// TIA Portal V20 export
DATA_BLOCK "ControlNodes"   // DB83
{ DB_Accessible_From_OPC_UA := 'FALSE' }
AUTHOR : ERsystem_FA2_DH. Kim
// stored: DBAccessibleFromOPCUA false, DBAccessibleFromWebserver false, MemoryReserve 100, Namespace Unit1.Em6
   VAR
      em { ExternalWritable := 'False'} : "LAF_typeEmControlNode";
      cm : Struct
         Interlock : Struct
            finalRollerFrontAxisX : "LER_typeAxisInterlock";
            finalRollerRearAxisX : "LER_typeAxisInterlock";
            mendrelAnodeFrontAxisY : "LER_typeAxisInterlock";
            mendrelAnodeFrontAxisZ : "LER_typeAxisInterlock";
            mendrelAnodeRearAxisY : "LER_typeAxisInterlock";
            mendrelAnodeRearAxisZ : "LER_typeAxisInterlock";
            mendrelCathodeFrontAxisY : "LER_typeAxisInterlock";
            mendrelCathodeFrontAxisZ : "LER_typeAxisInterlock";
            mendrelCathodeRearAxisY : "LER_typeAxisInterlock";
            mendrelCathodeRearAxisZ : "LER_typeAxisInterlock";
            stackTableAxisZ : "LER_typeAxisInterlock";
            stackTableOutFrontAxisZ : "LER_typeAxisInterlock";
            stackTableOutRearAxisZ : "LER_typeAxisInterlock";
            mendrelAnodeFrontClamp : "LER_typeTwoWayActInterlock";
            mendrelAnodeRearClamp : "LER_typeTwoWayActInterlock";
            mendrelCathodeFrontClamp : "LER_typeTwoWayActInterlock";
            mendrelCathodeRearClamp : "LER_typeTwoWayActInterlock";
            stackTableVaccum : "LER_typeTwoWayActInterlock";
            StackTableGapPadUpDown : "LER_typeTwoWayActInterlock";
         END_STRUCT;
         Command : Struct
            finalRollerFrontAxisX { S7_SetPoint := 'True'} : "LER_typeAxisCommand";
            finalRollerRearAxisX { S7_SetPoint := 'True'} : "LER_typeAxisCommand";
            mendrelAnodeFrontAxisY { S7_SetPoint := 'True'} : "LER_typeAxisCommand";
            mendrelAnodeFrontAxisZ { S7_SetPoint := 'True'} : "LER_typeAxisCommand";
            mendrelAnodeRearAxisY { S7_SetPoint := 'True'} : "LER_typeAxisCommand";
            mendrelAnodeRearAxisZ { S7_SetPoint := 'True'} : "LER_typeAxisCommand";
            mendrelCathodeFrontAxisY { S7_SetPoint := 'True'} : "LER_typeAxisCommand";
            mendrelCathodeFrontAxisZ { S7_SetPoint := 'True'} : "LER_typeAxisCommand";
            mendrelCathodeRearAxisY { S7_SetPoint := 'True'} : "LER_typeAxisCommand";
            mendrelCathodeRearAxisZ { S7_SetPoint := 'True'} : "LER_typeAxisCommand";
            stackTableAxisZ { S7_SetPoint := 'True'} : "LER_typeAxisCommand";
            stackTableOutFrontAxisZ { S7_SetPoint := 'True'} : "LER_typeAxisCommand";
            stackTableOutRearAxisZ { S7_SetPoint := 'True'} : "LER_typeAxisCommand";
         END_STRUCT;
         softCam { S7_SetPoint := 'True'} : "Unit1.type_emRelations_em6_SoftCam";
         brakeTest : Struct
            mendrelAnodeFrontAxisZ : "LER_typeBrakeTestEmControlNoeds";
            mendrelAnodeRearAxisZ : "LER_typeBrakeTestEmControlNoeds";
            mendrelCathodeFrontAxisZ : "LER_typeBrakeTestEmControlNoeds";
            mendrelCathodeRearAxisZ : "LER_typeBrakeTestEmControlNoeds";
            stackTableAxisZ : "LER_typeBrakeTestEmControlNoeds";
            stackTableOutFrontAxisZ : "LER_typeBrakeTestEmControlNoeds";
            stackTableOutRearAxisZ : "LER_typeBrakeTestEmControlNoeds";
         END_STRUCT;
         gearIn : Struct
            finalRollerAxisX : "LER_typeGearInControlNodes";
            stackTableOutAxisZ : "LER_typeGearInControlNodes";
            finalRollerFrontAxisX : Struct
               Execute : Bool;
               ContinuousUpdate : Bool;
               RatioNumerator : DInt;
               RatioDenominator : DInt;
               Acceleration : LReal;
               Deceleration : LReal;
               Jerk : LReal;
               PositionControlled : Bool;
               StartSync : Bool;
               InSync : Bool;
               ContinuousUpdateActive : Bool;
               Busy : Bool;
               CommandAborted : Bool;
               Error : Bool;
               ErrorId : Word;
            END_STRUCT;
            finalRollerRearAxisX : Struct
               Execute : Bool;
               ContinuousUpdate : Bool;
               RatioNumerator : DInt;
               RatioDenominator : DInt;
               Acceleration : LReal;
               Deceleration : LReal;
               Jerk : LReal;
               PositionControlled : Bool;
               StartSync : Bool;
               InSync : Bool;
               ContinuousUpdateActive : Bool;
               Busy : Bool;
               CommandAborted : Bool;
               Error : Bool;
               ErrorId : Word;
            END_STRUCT;
            stackTableOutFrontAxisZ : Struct
               Execute : Bool;
               ContinuousUpdate : Bool;
               RatioNumerator : DInt;
               RatioDenominator : DInt;
               Acceleration : LReal;
               Deceleration : LReal;
               Jerk : LReal;
               PositionControlled : Bool;
               StartSync : Bool;
               InSync : Bool;
               ContinuousUpdateActive : Bool;
               Busy : Bool;
               CommandAborted : Bool;
               Error : Bool;
               ErrorId : Word;
            END_STRUCT;
            stackTableOutRearAxisZ : Struct
               Execute : Bool;
               ContinuousUpdate : Bool;
               RatioNumerator : DInt;
               RatioDenominator : DInt;
               Acceleration : LReal;
               Deceleration : LReal;
               Jerk : LReal;
               PositionControlled : Bool;
               StartSync : Bool;
               InSync : Bool;
               ContinuousUpdateActive : Bool;
               Busy : Bool;
               CommandAborted : Bool;
               Error : Bool;
               ErrorId : Word;
            END_STRUCT;
         END_STRUCT;
         writeParameter : Struct
            finalRollerFrontAxisX : Struct
               Execute : Bool;
               ParameterNumber : DInt;
               Value { ExternalAccessible := 'False'; ExternalVisible := 'False'; ExternalWritable := 'False'} : LReal;
               Done : Bool;
               Busy : Bool;
               CommandAborted : Bool;
               Error : Bool;
               ErrorId : Word;
            END_STRUCT;
            finalRollerRearAxisX : Struct
               Execute : Bool;
               ParameterNumber : DInt;
               Value { ExternalAccessible := 'False'; ExternalVisible := 'False'; ExternalWritable := 'False'} : LReal;
               Done : Bool;
               Busy : Bool;
               CommandAborted : Bool;
               Error : Bool;
               ErrorId : Word;
            END_STRUCT;
            stackTableOutFrontAxisZ : Struct
               Execute : Bool;
               ParameterNumber : DInt;
               Value { ExternalAccessible := 'False'; ExternalVisible := 'False'; ExternalWritable := 'False'} : LReal;
               Done : Bool;
               Busy : Bool;
               CommandAborted : Bool;
               Error : Bool;
               ErrorId : Word;
            END_STRUCT;
            stackTableOutRearAxisZ : Struct
               Execute : Bool;
               ParameterNumber : DInt;
               Value { ExternalAccessible := 'False'; ExternalVisible := 'False'; ExternalWritable := 'False'} : LReal;
               Done : Bool;
               Busy : Bool;
               CommandAborted : Bool;
               Error : Bool;
               ErrorId : Word;
            END_STRUCT;
         END_STRUCT;
      END_STRUCT;
      stackTable : Struct
         jobs : "LAF_typeJobs";
         sequence { S7_SetPoint := 'True'} : "LAF_typeSequence";
         "step" { S7_SetPoint := 'True'} : "LER_typeStep";
         jobInterface : Struct
            homeJob1 : "LER_typeJobInterface";
            finalRollerJob12 : "LER_typeJobInterface";
            anodeMendrelJob22 : "LER_typeJobInterface";
            finalRollerJob13 : "LER_typeJobInterface";
            cathodeMendrelJob23 : "LER_typeJobInterface";
            visionJob30 : "LER_typeJobInterface";
            tableDownJob31 : "LER_typeJobInterface";
            unloadJob4 : "LER_typeJobInterface";
         END_STRUCT;
         preOperationCheck : Struct
            cathode : Bool;
            anode : Bool;
            Bool3 : Bool;
            Bool4 : Bool;
            Bool5 : Bool;
            Bool6 : Bool;
            Bool7 : Bool;
            Bool8 : Bool;
            Bool9 : Bool;
            Bool10 : Bool;
            Bool11 : Bool;
            Bool12 : Bool;
            Bool13 : Bool;
            Bool14 : Bool;
            Bool15 : Bool;
            Bool16 : Bool;
            Bool17 : Bool;
            Bool18 : Bool;
            Bool19 : Bool;
            Bool20 : Bool;
         END_STRUCT;
      END_STRUCT;
      gaugeRnR : Struct
         jobs : "LAF_typeJobs";
         sequence { S7_SetPoint := 'True'} : "LAF_typeSequence";
         "step" { S7_SetPoint := 'True'} : "LER_typeStep";
         jobInterface : Struct
            readyJob1 : "LER_typeJobInterface";
            vaccumJob2 : "LER_typeJobInterface";
            visionJob3 : "LER_typeJobInterface";
            blowJob4 : "LER_typeJobInterface";
         END_STRUCT;
         homeCheck : Struct
            home : Bool;
         END_STRUCT;
      END_STRUCT;
      emRelations : Struct
         em4 : Struct
            reqStackVaccum : Bool;
            reqStackBlow : Bool;
            donePnPUp : Bool;
            softCam : "Unit1.type_emRelations_em4_SoftCam";
         END_STRUCT;
         em5 : Struct
            reqStackVaccum : Bool;
            reqStackBlow : Bool;
            donePnPUp : Bool;
            softCam : "Unit1.type_emRelations_em5_SoftCam";
         END_STRUCT;
         em7 : Struct
            softCam : "Unit1.type_emRelations_em7_SoftCam";
         END_STRUCT;
      END_STRUCT;
      motionRelations : Struct
         commands : Struct
            null : Bool;
         END_STRUCT;
         monitoring : Struct
            null : Bool;
         END_STRUCT;
         config : Struct
            null : Bool;
         END_STRUCT;
      END_STRUCT;
      utility : Struct
         jobs : "LAF_typeJobs";
         sequence { S7_SetPoint := 'True'} : "LAF_typeSequence";
         "step" { S7_SetPoint := 'True'} : "LER_typeStep";
         jobInterface : Struct
            Job1 : "LER_typeJobInterface";
         END_STRUCT;
         homeCheck : Struct
            home : Bool;
         END_STRUCT;
      END_STRUCT;
      recipe : Struct
         anodeThickness : LReal;
         cathodeThickness : LReal;
         sepaThickenss : LReal;
         jellyRollThickness : LReal;
      END_STRUCT;
      parameters : Struct
         currentJellyRollThickness : LReal;
         currentStackCount : LReal;
         currentLastElectrode : LReal;   // 0 = Cathode / 1 = Anode
         finalRollerFrontHomeOffset : LReal;
         finalRollerRearHomeOffset : LReal;
         stackTableOutFrontHomeOffset : LReal;
         stackTableOutRearHomeOffset : LReal;
      END_STRUCT;
      cmStackTableElectrodeDetect { S7_SetPoint := 'True'} : "LBC_typeDigitalSignalControlNode";
   END_VAR
   VAR RETAIN
      cmMasterVirtualAxisX { ExternalVisible := 'False'; ExternalWritable := 'False'} : "LBC_typeAxis64PosControlNode";
   END_VAR
   VAR
      cmFinalRollerFrontAxisX { ExternalAccessible := 'False'; ExternalVisible := 'False'; ExternalWritable := 'False'; S7_SetPoint := 'True'} : "LBC_typeAxis64PosControlNode";
      cmFinalRollerRearAxisX { ExternalAccessible := 'False'; ExternalVisible := 'False'; ExternalWritable := 'False'; S7_SetPoint := 'True'} : "LBC_typeAxis64PosControlNode";
      cmMendrelAnodeFrontAxisY { ExternalAccessible := 'False'; ExternalVisible := 'False'; ExternalWritable := 'False'; S7_SetPoint := 'True'} : "LBC_typeAxis64PosControlNode";
      cmMendrelAnodeFrontAxisZ { ExternalAccessible := 'False'; ExternalVisible := 'False'; ExternalWritable := 'False'; S7_SetPoint := 'True'} : "LBC_typeAxis64PosControlNode";
      cmMendrelAnodeRearAxisY { ExternalAccessible := 'False'; ExternalVisible := 'False'; ExternalWritable := 'False'; S7_SetPoint := 'True'} : "LBC_typeAxis64PosControlNode";
      cmMendrelAnodeRearAxisZ { ExternalAccessible := 'False'; ExternalVisible := 'False'; ExternalWritable := 'False'; S7_SetPoint := 'True'} : "LBC_typeAxis64PosControlNode";
      cmMendrelCathodeFrontAxisY { ExternalAccessible := 'False'; ExternalVisible := 'False'; ExternalWritable := 'False'; S7_SetPoint := 'True'} : "LBC_typeAxis64PosControlNode";
      cmMendrelCathodeFrontAxisZ { ExternalAccessible := 'False'; ExternalVisible := 'False'; ExternalWritable := 'False'} : "LBC_typeAxis64PosControlNode";
      cmMendrelCathodeRearAxisY { ExternalAccessible := 'False'; ExternalVisible := 'False'; ExternalWritable := 'False'; S7_SetPoint := 'True'} : "LBC_typeAxis64PosControlNode";
      cmMendrelCathodeRearAxisZ { ExternalAccessible := 'False'; ExternalVisible := 'False'; ExternalWritable := 'False'; S7_SetPoint := 'True'} : "LBC_typeAxis64PosControlNode";
      cmStackTableAxisZ { ExternalAccessible := 'False'; ExternalVisible := 'False'; ExternalWritable := 'False'; S7_SetPoint := 'True'} : "LBC_typeAxis64PosControlNode";
      cmStackTableOutFrontAxisZ { ExternalAccessible := 'False'; ExternalVisible := 'False'; ExternalWritable := 'False'; S7_SetPoint := 'True'} : "LBC_typeAxis64PosControlNode";
      cmStackTableOutRearAxisZ { ExternalAccessible := 'False'; ExternalVisible := 'False'; ExternalWritable := 'False'; S7_SetPoint := 'True'} : "LBC_typeAxis64PosControlNode";
      cmMendrelAnodeFrontClamp { ExternalAccessible := 'False'; ExternalVisible := 'False'; ExternalWritable := 'False'; S7_SetPoint := 'True'} : "LBC_typeTwoWayActuatorControlNode";
      cmMendrelAnodeRearClamp { ExternalAccessible := 'False'; ExternalVisible := 'False'; ExternalWritable := 'False'; S7_SetPoint := 'True'} : "LBC_typeTwoWayActuatorControlNode";
      cmMendrelCathodeFrontClamp { ExternalAccessible := 'False'; ExternalVisible := 'False'; ExternalWritable := 'False'; S7_SetPoint := 'True'} : "LBC_typeTwoWayActuatorControlNode";
      cmMendrelCathodeRearClamp { ExternalAccessible := 'False'; ExternalVisible := 'False'; ExternalWritable := 'False'; S7_SetPoint := 'True'} : "LBC_typeTwoWayActuatorControlNode";
      cmStackTableVaccum { ExternalAccessible := 'False'; ExternalVisible := 'False'; ExternalWritable := 'False'; S7_SetPoint := 'True'} : "LBC_typeTwoWayActuatorControlNode";
      cmStackTableGapPadUpDown { ExternalAccessible := 'False'; ExternalVisible := 'False'; ExternalWritable := 'False'; S7_SetPoint := 'True'} : "LBC_typeTwoWayActuatorControlNode";
      cmStackGapVisionControllerInterface { ExternalAccessible := 'False'; ExternalVisible := 'False'; ExternalWritable := 'False'; S7_SetPoint := 'True'} : "LER_typeVisionControlNode";
   END_VAR
BEGIN
   em.commands.enable := FALSE;
   em.commands.acknowledge := FALSE;
   em.commands.disableAlarms := FALSE;
   em.commands.activateSimulation := FALSE;
   em.commands.home := FALSE;
   em.commands.moveToInitialPosition := FALSE;
   em.commands.directModeControl.current := 2;
   em.commands.directModeControl.production := FALSE;
   em.commands.directModeControl.maintenance := TRUE;
   em.commands.directModeControl.manual := FALSE;
   em.commands.directModeControl.nomode := FALSE;
   em.commands.directModeControl.sleep := FALSE;
   em.commands.directModeControl.deepsleep := FALSE;
   em.commands.directModeControl.userMode04 := FALSE;
   em.commands.directModeControl.userMode05 := FALSE;
   em.commands.directModeControl.userMode06 := FALSE;
   em.commands.directModeControl.userMode07 := FALSE;
   em.commands.directModeControl.userMode08 := FALSE;
   em.commands.directModeControl.userMode09 := FALSE;
   em.commands.directModeControl.userMode10 := FALSE;
   em.commands.directModeControl.userMode11 := FALSE;
   em.commands.directModeControl.userMode12 := FALSE;
   em.commands.directModeControl.userMode13 := FALSE;
   em.commands.directStateControl.current := 2;
   em.commands.directStateControl.clearing := FALSE;
   em.commands.directStateControl.stopped := TRUE;
   em.commands.directStateControl.starting := FALSE;
   em.commands.directStateControl.idle := FALSE;
   em.commands.directStateControl.suspended := FALSE;
   em.commands.directStateControl.execute := FALSE;
   em.commands.directStateControl.stopping := FALSE;
   em.commands.directStateControl.aborting := FALSE;
   em.commands.directStateControl.aborted := FALSE;
   em.commands.directStateControl.holding := FALSE;
   em.commands.directStateControl.held := FALSE;
   em.commands.directStateControl.unholding := FALSE;
   em.commands.directStateControl.suspending := FALSE;
   em.commands.directStateControl.unsuspending := FALSE;
   em.commands.directStateControl.resetting := FALSE;
   em.commands.directStateControl.completing := FALSE;
   em.commands.directStateControl.complete := FALSE;
   em.status.enabled := FALSE;
   em.status.acknowledgeActive := FALSE;
   em.status.alarmsDisabled := FALSE;
   em.status.simulationActive := FALSE;
   em.status.safetyReleased := TRUE;
   em.status.initialized := FALSE;
   em.status.homed := FALSE;
   em.status.safeState := FALSE;
   em.status.stateComplete := TRUE;
   cm.gearIn.finalRollerAxisX.command.ratioNumerator := 1;
   cm.gearIn.finalRollerAxisX.command.ratioDenominator := 1;
   cm.gearIn.finalRollerAxisX.command.acceleration := -1.0;
   cm.gearIn.finalRollerAxisX.command.deceleration := -1.0;
   cm.gearIn.finalRollerAxisX.command.positionControlled := TRUE;
   cm.gearIn.stackTableOutAxisZ.command.ratioNumerator := 1;
   cm.gearIn.stackTableOutAxisZ.command.ratioDenominator := 1;
   cm.gearIn.stackTableOutAxisZ.command.acceleration := -1.0;
   cm.gearIn.stackTableOutAxisZ.command.deceleration := -1.0;
   cm.gearIn.stackTableOutAxisZ.command.positionControlled := TRUE;
   // stackTable."step".action1[101] : Step[101] : JOB[1] Condition
   // stackTable."step".action1[110] : Step[110] : StackTableOut Z-Axis Wait(=Down) Pos
   // stackTable."step".action1[120] : Step[120] : GapPad Up
   // stackTable."step".action1[130] : Step[130] : A,C.Mendrel Clamp Work Pos [Request Check]
   // stackTable."step".action1[140] : Step[140] : C.Mendrel Y,Z-Axis Wait Pos
   // stackTable."step".action1[141] : Step[141] : C.Mendrel Y,Z-Axis Work Pos
   // stackTable."step".action1[142] : Step[142] : Stack Table → Anode Main P&P [Clamp Done]
   // stackTable."step".action1[150] : Step[150] : FinalRoller X-Axis Anode Pos [Request Check]
   // stackTable."step".action1[160] : Step[160] : A.Mendrel Y,Z-Axis Wait Pos
   // stackTable."step".action1[161] : Step[161] : A.Mendrel Y,Z-Axis Work Pos
   // stackTable."step".action1[162] : Step[162] : Stack Table → Cathode Main P&P [Clamp Done]
   // stackTable."step".action1[170] : Step[170] : FinalRoller X-Axis Cathode Pos [Request Check]
   // stackTable."step".action1[180] : Step[180] : C.Mendrel Y,Z-Axis Wait Pos
   // stackTable."step".action1[181] : Step[181] : C.Mendrel Y,Z-Axis Work Pos
   // stackTable."step".action1[182] : Step[182] : Stack Table → Anode Main P&P [Clamp Done]
   // stackTable."step".action1[183] : Step[183] : C.Mendrel Y,Z-Axis Wait Pos
   // stackTable."step".action1[184] : Step[184] : C.Mendrel Y,Z-Axis Work Pos
   // stackTable."step".action1[185] : Step[185] : Stack Table → Anode Main P&P [Clamp Done]
   // stackTable."step".action1[190] : Step[190] : Job [1] Step End
   // stackTable."step".action1[201] : Step[201] : JOB[2] Condition
   // stackTable."step".action1[210] : Step[210] : FinalRoller X-Axis Anode Pos [Unloading Ready Check]
   // stackTable."step".action1[220] : Step[220] : A.Mendrel Y,Z-Axis Wait Pos
   // stackTable."step".action1[221] : Step[221] : A.Mendrel Y,Z-Axis Work Pos
   // stackTable."step".action1[222] : Step[222] : Stack Table → Cathode Main P&P [Clamp Done]
   // stackTable."step".action1[280] : Step[280] : Stack Table Z-Axis Work(=Down) Pos
   // stackTable."step".action1[290] : Step[290] : JOB[2] Condition
   // stackTable."step".action1[301] : Step[301] : JOB[3] Condition
   // stackTable."step".action1[310] : Step[310] : FinalRoller X-Axis Cathode Pos [Unloading Ready Check]
   // stackTable."step".action1[320] : Step[320] : C.Mendrel Y,Z-Axis Wait Pos
   // stackTable."step".action1[321] : Step[321] : C.Mendrel Y,Z-Axis Work Pos
   // stackTable."step".action1[322] : Step[322] : Stack Table → Anode Main P&P [Clamp Done]
   // stackTable."step".action1[380] : Step[380] : Stack Table Z-Axis Work(=Down) Pos
   // stackTable."step".action1[390] : Step[390] : JOB[3] Condition
   // stackTable."step".action1[401] : Step[401] : JOB[4] Condition
   // stackTable."step".action1[420] : Step[420] : GapPad Down
   // stackTable."step".action1[421] : Step[421] : Stack Table → Sepa Stack P&P [Unload Request]
   // stackTable."step".action1[430] : Step[430] : A,C.Mendrel Y,Z-Axis Wait Pos
   // stackTable."step".action1[431] : Step[431] : Stack Table → Sepa Stack P&P [Unclamp Done]
   // stackTable."step".action1[440] : Step[440] : A,C.Mendrel Y,Z-Axis Work Pos
   // stackTable."step".action1[441] : Step[441] : Stack Table → Sepa Stack P&P [Clamp Done]
   // stackTable."step".action1[450] : Step[450] : GapPad Up
   // stackTable."step".action1[480] : Step[480] : StackTableOut Z-Axis Wait(=Down) Pos
   // stackTable."step".action1[490] : Step[490] : JOB[4] Condition
   // stackTable."step".transition1[101] : Step[101] : JOB[1] Condition
   // stackTable."step".transition1[110] : Step[110] : StackTableOut Z-Axis Wait(=Down) Pos
   // stackTable."step".transition1[120] : Step[120] : GapPad Up
   // stackTable."step".transition1[130] : Step[130] : A,C.Mendrel Clamp Work Pos [Request Check]
   // stackTable."step".transition1[140] : Step[140] : C.Mendrel Y,Z-Axis Wait Pos
   // stackTable."step".transition1[141] : Step[141] : C.Mendrel Y,Z-Axis Work Pos
   // stackTable."step".transition1[142] : Step[142] : Stack Table → Anode Main P&P [Clamp Done]
   // stackTable."step".transition1[150] : Step[150] : FinalRoller X-Axis Anode Pos [Request Check]
   // stackTable."step".transition1[160] : Step[160] : A.Mendrel Y,Z-Axis Wait Pos
   // stackTable."step".transition1[161] : Step[161] : A.Mendrel Y,Z-Axis Work Pos
   // stackTable."step".transition1[162] : Step[162] : Stack Table → Cathode Main P&P [Clamp Done]
   // stackTable."step".transition1[170] : Step[170] : FinalRoller X-Axis Cathode Pos [Request Check]
   // stackTable."step".transition1[180] : Step[180] : C.Mendrel Y,Z-Axis Wait Pos
   // stackTable."step".transition1[181] : Step[181] : C.Mendrel Y,Z-Axis Work Pos
   // stackTable."step".transition1[182] : Step[182] : Stack Table → Anode Main P&P [Clamp Done]
   // stackTable."step".transition1[183] : Step[183] : C.Mendrel Y,Z-Axis Wait Pos
   // stackTable."step".transition1[184] : Step[184] : C.Mendrel Y,Z-Axis Work Pos
   // stackTable."step".transition1[185] : Step[185] : Stack Table → Anode Main P&P [Clamp Done]
   // stackTable."step".transition1[190] : Step[190] : Job [1] Step End
   // stackTable."step".transition1[201] : Step[201] : JOB[2] Condition
   // stackTable."step".transition1[210] : Step[210] : FinalRoller X-Axis Anode Pos [Unloading Ready Check]
   // stackTable."step".transition1[220] : Step[220] : A.Mendrel Y,Z-Axis Wait Pos
   // stackTable."step".transition1[221] : Step[221] : A.Mendrel Y,Z-Axis Work Pos
   // stackTable."step".transition1[222] : Step[222] : Stack Table → Cathode Main P&P [Clamp Done]
   // stackTable."step".transition1[280] : Step[280] : Stack Table Z-Axis Work(=Down) Pos
   // stackTable."step".transition1[290] : Step[290] : JOB[2] Condition
   // stackTable."step".transition1[301] : Step[301] : JOB[3] Condition
   // stackTable."step".transition1[310] : Step[310] : FinalRoller X-Axis Cathode Pos [Unloading Ready Check]
   // stackTable."step".transition1[320] : Step[320] : C.Mendrel Y,Z-Axis Wait Pos
   // stackTable."step".transition1[321] : Step[321] : C.Mendrel Y,Z-Axis Work Pos
   // stackTable."step".transition1[322] : Step[322] : Stack Table → Anode Main P&P [Clamp Done]
   // stackTable."step".transition1[380] : Step[380] : Stack Table Z-Axis Work(=Down) Pos
   // stackTable."step".transition1[390] : Step[390] : JOB[3] Condition
   // stackTable."step".transition1[401] : Step[401] : JOB[4] Condition
   // stackTable."step".transition1[420] : Step[420] : GapPad Down
   // stackTable."step".transition1[421] : Step[421] : Stack Table → Sepa Stack P&P [Unload Request]
   // stackTable."step".transition1[430] : Step[430] : A,C.Mendrel Y,Z-Axis Wait Pos
   // stackTable."step".transition1[431] : Step[431] : Stack Table → Sepa Stack P&P [Unclamp Done]
   // stackTable."step".transition1[440] : Step[440] : A,C.Mendrel Y,Z-Axis Work Pos
   // stackTable."step".transition1[441] : Step[441] : Stack Table → Sepa Stack P&P [Clamp Done]
   // stackTable."step".transition1[450] : Step[450] : GapPad Up
   // stackTable."step".transition1[480] : Step[480] : StackTableOut Z-Axis Wait(=Down) Pos
   // stackTable."step".transition1[490] : Step[490] : JOB[4] Condition
   // gaugeRnR."step".action1[101] : Step[101] : JOB[1] Condition
   // gaugeRnR."step".action1[110] : Step[110] : Mendrel Z-Axis Up
   // gaugeRnR."step".action1[120] : Step[120] : Mendrel Y-Axis Backward
   // gaugeRnR."step".action1[130] : Step[130] : StackTable Blow
   // gaugeRnR."step".action1[190] : Step[190] : Job [1] Step End
   // gaugeRnR."step".action1[201] : Step[201] : JOB[2] Condition
   // gaugeRnR."step".action1[210] : Step[210] : StackTable Vaccum
   // gaugeRnR."step".action1[290] : Step[290] Job [2] Step End
   // gaugeRnR."step".action1[301] : Step[301] : JOB[3] Condition
   // gaugeRnR."step".action1[310] : Step[310] : Anode Vision Start
   // gaugeRnR."step".action1[330] : Step[330] : Cathode Vision Start
   // gaugeRnR."step".action1[390] : Step[390] Job [3] Step End
   // gaugeRnR."step".action1[401] : Step[401] : JOB[4] Condition
   // gaugeRnR."step".action1[410] : Step[410] : StackTable Blow
   // gaugeRnR."step".action1[490] : Step[490] Job [4] Step End
   // gaugeRnR."step".transition1[101] : Step[101] : JOB[1] Condition
   // gaugeRnR."step".transition1[110] : Step[110] : Mendrel Z-Axis Up
   // gaugeRnR."step".transition1[120] : Step[120] : Mendrel Y-Axis Backward
   // gaugeRnR."step".transition1[130] : Step[130] : StackTable Blow
   // gaugeRnR."step".transition1[190] : Step[190] : Job [1] Step End
   // gaugeRnR."step".transition1[201] : Step[201] : JOB[2] Condition
   // gaugeRnR."step".transition1[210] : Step[210] : StackTable Vaccum
   // gaugeRnR."step".transition1[290] : Step[290] Job [2] Step End
   // gaugeRnR."step".transition1[301] : Step[301] : JOB[3] Condition
   // gaugeRnR."step".transition1[310] : Step[310] : Anode Vision Start
   // gaugeRnR."step".transition1[330] : Step[330] : Cathode Vision Start
   // gaugeRnR."step".transition1[390] : Step[390] Job [3] Step End
   // gaugeRnR."step".transition1[401] : Step[401] : JOB[4] Condition
   // gaugeRnR."step".transition1[410] : Step[410] : StackTable Blow
   // gaugeRnR."step".transition1[490] : Step[490] Job [4] Step End
   cmStackTableElectrodeDetect.commands.reset := FALSE;
   cmStackTableElectrodeDetect.commands.simulation := FALSE;
   cmStackTableElectrodeDetect.commands.quality := TRUE;
   cmStackTableElectrodeDetect.monitoring.valid := TRUE;
   cmStackTableElectrodeDetect.monitoring.busy := TRUE;
   cmStackTableElectrodeDetect.monitoring.error := FALSE;
   cmStackTableElectrodeDetect.monitoring.status := 16#0000;
   cmStackTableElectrodeDetect.monitoring.risingEdge := FALSE;
   cmStackTableElectrodeDetect.monitoring.fallingEdge := FALSE;
   cmStackTableElectrodeDetect.monitoring.processValue := FALSE;
   cmFinalRollerFrontAxisX.commandConfiguration.generalSettings.stopOnError := TRUE;
   cmFinalRollerFrontAxisX.commandConfiguration.generalSettings.resetWithRestart := FALSE;
   cmFinalRollerFrontAxisX.commandConfiguration.generalSettings.abortWaitingSyncCmd := TRUE;
   cmFinalRollerFrontAxisX.commandConfiguration.power.startMode := 1;
   cmFinalRollerFrontAxisX.commandConfiguration.power.stopMode := 0;
   cmFinalRollerFrontAxisX.commandConfiguration.power.syncMotionSimulation := FALSE;
   cmFinalRollerFrontAxisX.commandConfiguration.power.syncMotionSimulationExtendedMode := -1;
   cmFinalRollerFrontAxisX.commandConfiguration.jog.velocity := 0.0;
   cmFinalRollerFrontAxisX.commandConfiguration.jog.acceleration := -1.0;
   cmFinalRollerFrontAxisX.commandConfiguration.jog.deceleration := -1.0;
   cmFinalRollerFrontAxisX.commandConfiguration.jog.jerk := -1.0;
   cmFinalRollerFrontAxisX.commandConfiguration.jog.positionControlled := TRUE;
   cmFinalRollerFrontAxisX.commandConfiguration.jog.increment := 0.0;
   cmFinalRollerFrontAxisX.commandConfiguration.jog.mode := 0;
   cmFinalRollerFrontAxisX.commandConfiguration.moveVelocity.velocity := 0.0;
   cmFinalRollerFrontAxisX.commandConfiguration.moveVelocity.acceleration := -1.0;
   cmFinalRollerFrontAxisX.commandConfiguration.moveVelocity.deceleration := -1.0;
   cmFinalRollerFrontAxisX.commandConfiguration.moveVelocity.jerk := -1.0;
   cmFinalRollerFrontAxisX.commandConfiguration.moveVelocity.direction := 0;
   cmFinalRollerFrontAxisX.commandConfiguration.moveVelocity.positionControlled := TRUE;
   cmFinalRollerFrontAxisX.commandConfiguration.moveVelocity.velocityChangeOnTheFly := FALSE;
   cmFinalRollerFrontAxisX.commandConfiguration.stop.deceleration := -1.0;
   cmFinalRollerFrontAxisX.commandConfiguration.stop.jerk := -1.0;
   cmFinalRollerFrontAxisX.commandConfiguration.stop.abortAcceleration := FALSE;
   cmFinalRollerFrontAxisX.commandConfiguration.fastStop.deceleration := -1.0;
   cmFinalRollerFrontAxisX.commandConfiguration.fastStop.jerk := -1.0;
   cmFinalRollerFrontAxisX.commandConfiguration.fastStop.abortAcceleration := FALSE;
   cmFinalRollerFrontAxisX.commandConfiguration.fastStop.replaceStopPossible := FALSE;
   cmFinalRollerFrontAxisX.commandConfiguration.torqueLimiting.limit := -1.0;
   cmFinalRollerFrontAxisX.commandConfiguration.torqueLimiting.mode := 0;
   // cmFinalRollerFrontAxisX.commandConfiguration.homing.mode : Homing Mode
   cmFinalRollerFrontAxisX.commandConfiguration.posAbsolute.position := 0.0;
   cmFinalRollerFrontAxisX.commandConfiguration.posAbsolute.velocity := -1.0;
   cmFinalRollerFrontAxisX.commandConfiguration.posAbsolute.acceleration := -1.0;
   cmFinalRollerFrontAxisX.commandConfiguration.posAbsolute.deceleration := -1.0;
   cmFinalRollerFrontAxisX.commandConfiguration.posAbsolute.jerk := -1.0;
   cmFinalRollerFrontAxisX.commandConfiguration.posAbsolute.direction := 1;
   cmFinalRollerFrontAxisX.commandConfiguration.posAbsolute.positionChangeOnTheFly := FALSE;
   cmFinalRollerFrontAxisX.commandConfiguration.posAbsolute.velocityChangeOnTheFly := FALSE;
   cmFinalRollerFrontAxisX.commandConfiguration.posSuperimposed.distance := 0.0;
   cmFinalRollerFrontAxisX.commandConfiguration.posSuperimposed.velocityDiff := -1.0;
   cmFinalRollerFrontAxisX.commandConfiguration.posSuperimposed.acceleration := -1.0;
   cmFinalRollerFrontAxisX.commandConfiguration.posSuperimposed.deceleration := -1.0;
   cmFinalRollerFrontAxisX.commandConfiguration.posSuperimposed.jerk := -1.0;
   cmFinalRollerFrontAxisX.commandConfiguration.posSuperimposed.direction := 0;
   cmFinalRollerFrontAxisX.commandConfiguration.haltSuperimposed.deceleration := -1.0;
   cmFinalRollerFrontAxisX.commandConfiguration.haltSuperimposed.jerk := -1.0;
   cmFinalRollerFrontAxisX.commandConfiguration.haltSuperimposed.abortAcceleration := FALSE;
   cmFinalRollerFrontAxisX.commandConfiguration.gearInRelative.ratioNumerator := 1;
   cmFinalRollerFrontAxisX.commandConfiguration.gearInRelative.ratioDenominator := 1;
   cmFinalRollerFrontAxisX.commandConfiguration.gearInRelative.acceleration := -1.0;
   cmFinalRollerFrontAxisX.commandConfiguration.gearInRelative.deceleration := -1.0;
   cmFinalRollerFrontAxisX.commandConfiguration.gearInRelative.jerk := -1.0;
   cmFinalRollerFrontAxisX.commandConfiguration.gearInRelative.ratioChangeOnTheFly := FALSE;
   cmFinalRollerFrontAxisX.commandConfiguration.gearInAbsolute.ratioNumerator := 1;
   cmFinalRollerFrontAxisX.commandConfiguration.gearInAbsolute.ratioDenominator := 1;
   cmFinalRollerFrontAxisX.commandConfiguration.gearInAbsolute.masterSyncPosition := 0.0;
   cmFinalRollerFrontAxisX.commandConfiguration.gearInAbsolute.slaveSyncPosition := 0.0;
   cmFinalRollerFrontAxisX.commandConfiguration.gearInAbsolute.syncProfileReference := 1;
   cmFinalRollerFrontAxisX.commandConfiguration.gearInAbsolute.masterStartDistance := 0.0;
   cmFinalRollerFrontAxisX.commandConfiguration.gearInAbsolute.velocity := -1.0;
   cmFinalRollerFrontAxisX.commandConfiguration.gearInAbsolute.acceleration := -1.0;
   cmFinalRollerFrontAxisX.commandConfiguration.gearInAbsolute.deceleration := -1.0;
   cmFinalRollerFrontAxisX.commandConfiguration.gearInAbsolute.jerk := -1.0;
   cmFinalRollerFrontAxisX.commandConfiguration.gearInAbsolute.syncDirection := 1;
   cmFinalRollerFrontAxisX.commandConfiguration.gearInAbsolute.ratioChangeOnTheFly := FALSE;
   cmFinalRollerFrontAxisX.commandConfiguration.gearInVelocity.continuousUpdate := FALSE;
   cmFinalRollerFrontAxisX.commandConfiguration.gearInVelocity.ratioNumerator := 1;
   cmFinalRollerFrontAxisX.commandConfiguration.gearInVelocity.ratioDenominator := 1;
   cmFinalRollerFrontAxisX.commandConfiguration.gearInVelocity.acceleration := -1.0;
   cmFinalRollerFrontAxisX.commandConfiguration.gearInVelocity.deceleration := -1.0;
   cmFinalRollerFrontAxisX.commandConfiguration.gearInVelocity.jerk := -1.0;
   cmFinalRollerFrontAxisX.commandConfiguration.gearInVelocity.positionControlled := FALSE;
   cmFinalRollerFrontAxisX.commandConfiguration.camIn.masterOffset := 0.0;
   cmFinalRollerFrontAxisX.commandConfiguration.camIn.slaveOffset := 0.0;
   cmFinalRollerFrontAxisX.commandConfiguration.camIn.masterScaling := 1.0;
   cmFinalRollerFrontAxisX.commandConfiguration.camIn.slaveScaling := 1.0;
   cmFinalRollerFrontAxisX.commandConfiguration.camIn.masterSyncPosition := 0.0;
   cmFinalRollerFrontAxisX.commandConfiguration.camIn.syncProfileReference := 1;
   cmFinalRollerFrontAxisX.commandConfiguration.camIn.masterStartDistance := 0.0;
   cmFinalRollerFrontAxisX.commandConfiguration.camIn.velocity := -1.0;
   cmFinalRollerFrontAxisX.commandConfiguration.camIn.acceleration := -1.0;
   cmFinalRollerFrontAxisX.commandConfiguration.camIn.deceleration := -1.0;
   cmFinalRollerFrontAxisX.commandConfiguration.camIn.jerk := -1.0;
   cmFinalRollerFrontAxisX.commandConfiguration.camIn.applicationMode := 0;
   cmFinalRollerFrontAxisX.commandConfiguration.camIn.syncDirection := 1;
   cmFinalRollerFrontAxisX.commandConfiguration.gearOutCamOut.slavePosition := 0.0;
   cmFinalRollerFrontAxisX.commandConfiguration.gearOutCamOut.syncProfileReference := 1;
   cmFinalRollerFrontAxisX.commandConfiguration.gearOutCamOut.masterStopDistance := 0.0;
   cmFinalRollerFrontAxisX.commandConfiguration.gearOutCamOut.deceleration := -1.0;
   cmFinalRollerFrontAxisX.commandConfiguration.gearOutCamOut.jerk := -1.0;
   cmFinalRollerFrontAxisX.commandConfiguration.gearOutCamOut.syncOutDirection := 3;
   cmFinalRollerFrontAxisX.commandConfiguration.gearOutCamOut.gearOutCamOutMode := -1;
   cmFinalRollerFrontAxisX.commandConfiguration.phasing.phaseShift := 0.0;
   cmFinalRollerFrontAxisX.commandConfiguration.phasing.velocity := -1.0;
   cmFinalRollerFrontAxisX.commandConfiguration.phasing.acceleration := -1.0;
   cmFinalRollerFrontAxisX.commandConfiguration.phasing.deceleration := -1.0;
   cmFinalRollerFrontAxisX.commandConfiguration.phasing.jerk := -1.0;
   cmFinalRollerFrontAxisX.commandConfiguration.phasing.profileReference := 0;
   cmFinalRollerFrontAxisX.commandConfiguration.phasing.phasingDistance := 0.0;
   cmFinalRollerFrontAxisX.commandConfiguration.phasing.startPosition := 0.0;
   cmFinalRollerFrontAxisX.commandConfiguration.phasing.direction := 3;
   cmFinalRollerFrontAxisX.commandConfiguration.phasing.phaseAbsolute := TRUE;
   cmFinalRollerFrontAxisX.commandConfiguration.phasing.phaseShiftChangeOnTheFly := FALSE;
   cmFinalRollerFrontAxisX.commandConfiguration.offset.offset := 0.0;
   cmFinalRollerFrontAxisX.commandConfiguration.offset.profileReference := 1;
   cmFinalRollerFrontAxisX.commandConfiguration.offset.offsetDistance := 0.0;
   cmFinalRollerFrontAxisX.commandConfiguration.offset.startPosition := 0.0;
   cmFinalRollerFrontAxisX.commandConfiguration.offset.direction := 3;
   cmFinalRollerFrontAxisX.commandConfiguration.offset.offsetAbsolute := TRUE;
   cmFinalRollerFrontAxisX.commandConfiguration.offset.offsetChangeOnTheFly := FALSE;
   cmMendrelAnodeFrontAxisY.commandConfiguration.generalSettings.stopOnError := TRUE;
   cmMendrelAnodeFrontAxisY.commandConfiguration.generalSettings.resetWithRestart := FALSE;
   cmMendrelAnodeFrontAxisY.commandConfiguration.generalSettings.abortWaitingSyncCmd := TRUE;
   cmMendrelAnodeFrontAxisY.commandConfiguration.power.startMode := 1;
   cmMendrelAnodeFrontAxisY.commandConfiguration.power.stopMode := 0;
   cmMendrelAnodeFrontAxisY.commandConfiguration.power.syncMotionSimulation := FALSE;
   cmMendrelAnodeFrontAxisY.commandConfiguration.power.syncMotionSimulationExtendedMode := -1;
   cmMendrelAnodeFrontAxisY.commandConfiguration.jog.velocity := 0.0;
   cmMendrelAnodeFrontAxisY.commandConfiguration.jog.acceleration := -1.0;
   cmMendrelAnodeFrontAxisY.commandConfiguration.jog.deceleration := -1.0;
   cmMendrelAnodeFrontAxisY.commandConfiguration.jog.jerk := -1.0;
   cmMendrelAnodeFrontAxisY.commandConfiguration.jog.positionControlled := TRUE;
   cmMendrelAnodeFrontAxisY.commandConfiguration.jog.increment := 0.0;
   cmMendrelAnodeFrontAxisY.commandConfiguration.jog.mode := 0;
   cmMendrelAnodeFrontAxisY.commandConfiguration.moveVelocity.velocity := 0.0;
   cmMendrelAnodeFrontAxisY.commandConfiguration.moveVelocity.acceleration := -1.0;
   cmMendrelAnodeFrontAxisY.commandConfiguration.moveVelocity.deceleration := -1.0;
   cmMendrelAnodeFrontAxisY.commandConfiguration.moveVelocity.jerk := -1.0;
   cmMendrelAnodeFrontAxisY.commandConfiguration.moveVelocity.direction := 0;
   cmMendrelAnodeFrontAxisY.commandConfiguration.moveVelocity.positionControlled := TRUE;
   cmMendrelAnodeFrontAxisY.commandConfiguration.moveVelocity.velocityChangeOnTheFly := FALSE;
   cmMendrelAnodeFrontAxisY.commandConfiguration.stop.deceleration := -1.0;
   cmMendrelAnodeFrontAxisY.commandConfiguration.stop.jerk := -1.0;
   cmMendrelAnodeFrontAxisY.commandConfiguration.stop.abortAcceleration := FALSE;
   cmMendrelAnodeFrontAxisY.commandConfiguration.fastStop.deceleration := -1.0;
   cmMendrelAnodeFrontAxisY.commandConfiguration.fastStop.jerk := -1.0;
   cmMendrelAnodeFrontAxisY.commandConfiguration.fastStop.abortAcceleration := FALSE;
   cmMendrelAnodeFrontAxisY.commandConfiguration.fastStop.replaceStopPossible := FALSE;
   cmMendrelAnodeFrontAxisY.commandConfiguration.torqueLimiting.limit := -1.0;
   cmMendrelAnodeFrontAxisY.commandConfiguration.torqueLimiting.mode := 0;
   cmMendrelAnodeFrontAxisY.commandConfiguration.homing.position := 0.0;
   cmMendrelAnodeFrontAxisY.commandConfiguration.homing.mode := 0;
   cmMendrelAnodeFrontAxisY.commandConfiguration.homing.sensor := 0;
   cmMendrelAnodeFrontAxisY.commandConfiguration.homing.extendedMode := -1;
   cmMendrelAnodeFrontAxisY.commandConfiguration.homing.extendedModeTorqueLimit := 0.0;
   cmMendrelAnodeFrontAxisY.commandConfiguration.homing.extendedModeTargetPosition := 0.0;
   cmMendrelAnodeFrontAxisY.commandConfiguration.posRelative.distance := 0.0;
   cmMendrelAnodeFrontAxisY.commandConfiguration.posRelative.velocity := -1.0;
   cmMendrelAnodeFrontAxisY.commandConfiguration.posRelative.acceleration := -1.0;
   cmMendrelAnodeFrontAxisY.commandConfiguration.posRelative.deceleration := -1.0;
   cmMendrelAnodeFrontAxisY.commandConfiguration.posRelative.jerk := -1.0;
   cmMendrelAnodeFrontAxisY.commandConfiguration.posRelative.direction := 0;
   cmMendrelAnodeFrontAxisY.commandConfiguration.posAbsolute.position := 0.0;
   cmMendrelAnodeFrontAxisY.commandConfiguration.posAbsolute.velocity := -1.0;
   cmMendrelAnodeFrontAxisY.commandConfiguration.posAbsolute.acceleration := -1.0;
   cmMendrelAnodeFrontAxisY.commandConfiguration.posAbsolute.deceleration := -1.0;
   cmMendrelAnodeFrontAxisY.commandConfiguration.posAbsolute.jerk := -1.0;
   cmMendrelAnodeFrontAxisY.commandConfiguration.posAbsolute.direction := 1;
   cmMendrelAnodeFrontAxisY.commandConfiguration.posAbsolute.positionChangeOnTheFly := FALSE;
   cmMendrelAnodeFrontAxisY.commandConfiguration.posAbsolute.velocityChangeOnTheFly := FALSE;
   cmMendrelAnodeFrontAxisY.commandConfiguration.posSuperimposed.distance := 0.0;
   cmMendrelAnodeFrontAxisY.commandConfiguration.posSuperimposed.velocityDiff := -1.0;
   cmMendrelAnodeFrontAxisY.commandConfiguration.posSuperimposed.acceleration := -1.0;
   cmMendrelAnodeFrontAxisY.commandConfiguration.posSuperimposed.deceleration := -1.0;
   cmMendrelAnodeFrontAxisY.commandConfiguration.posSuperimposed.jerk := -1.0;
   cmMendrelAnodeFrontAxisY.commandConfiguration.posSuperimposed.direction := 0;
   cmMendrelAnodeFrontAxisY.commandConfiguration.haltSuperimposed.deceleration := -1.0;
   cmMendrelAnodeFrontAxisY.commandConfiguration.haltSuperimposed.jerk := -1.0;
   cmMendrelAnodeFrontAxisY.commandConfiguration.haltSuperimposed.abortAcceleration := FALSE;
   cmMendrelAnodeFrontAxisY.commandConfiguration.gearInRelative.ratioNumerator := 1;
   cmMendrelAnodeFrontAxisY.commandConfiguration.gearInRelative.ratioDenominator := 1;
   cmMendrelAnodeFrontAxisY.commandConfiguration.gearInRelative.acceleration := -1.0;
   cmMendrelAnodeFrontAxisY.commandConfiguration.gearInRelative.deceleration := -1.0;
   cmMendrelAnodeFrontAxisY.commandConfiguration.gearInRelative.jerk := -1.0;
   cmMendrelAnodeFrontAxisY.commandConfiguration.gearInRelative.ratioChangeOnTheFly := FALSE;
   cmMendrelAnodeFrontAxisY.commandConfiguration.gearInAbsolute.ratioNumerator := 1;
   cmMendrelAnodeFrontAxisY.commandConfiguration.gearInAbsolute.ratioDenominator := 1;
   cmMendrelAnodeFrontAxisY.commandConfiguration.gearInAbsolute.masterSyncPosition := 0.0;
   cmMendrelAnodeFrontAxisY.commandConfiguration.gearInAbsolute.slaveSyncPosition := 0.0;
   cmMendrelAnodeFrontAxisY.commandConfiguration.gearInAbsolute.syncProfileReference := 1;
   cmMendrelAnodeFrontAxisY.commandConfiguration.gearInAbsolute.masterStartDistance := 0.0;
   cmMendrelAnodeFrontAxisY.commandConfiguration.gearInAbsolute.velocity := -1.0;
   cmMendrelAnodeFrontAxisY.commandConfiguration.gearInAbsolute.acceleration := -1.0;
   cmMendrelAnodeFrontAxisY.commandConfiguration.gearInAbsolute.deceleration := -1.0;
   cmMendrelAnodeFrontAxisY.commandConfiguration.gearInAbsolute.jerk := -1.0;
   cmMendrelAnodeFrontAxisY.commandConfiguration.gearInAbsolute.syncDirection := 1;
   cmMendrelAnodeFrontAxisY.commandConfiguration.gearInAbsolute.ratioChangeOnTheFly := FALSE;
   cmMendrelAnodeFrontAxisY.commandConfiguration.gearInVelocity.continuousUpdate := FALSE;
   cmMendrelAnodeFrontAxisY.commandConfiguration.gearInVelocity.ratioNumerator := 1;
   cmMendrelAnodeFrontAxisY.commandConfiguration.gearInVelocity.ratioDenominator := 1;
   cmMendrelAnodeFrontAxisY.commandConfiguration.gearInVelocity.acceleration := -1.0;
   cmMendrelAnodeFrontAxisY.commandConfiguration.gearInVelocity.deceleration := -1.0;
   cmMendrelAnodeFrontAxisY.commandConfiguration.gearInVelocity.jerk := -1.0;
   cmMendrelAnodeFrontAxisY.commandConfiguration.gearInVelocity.positionControlled := FALSE;
   cmMendrelAnodeFrontAxisY.commandConfiguration.camIn.masterOffset := 0.0;
   cmMendrelAnodeFrontAxisY.commandConfiguration.camIn.slaveOffset := 0.0;
   cmMendrelAnodeFrontAxisY.commandConfiguration.camIn.masterScaling := 1.0;
   cmMendrelAnodeFrontAxisY.commandConfiguration.camIn.slaveScaling := 1.0;
   cmMendrelAnodeFrontAxisY.commandConfiguration.camIn.masterSyncPosition := 0.0;
   cmMendrelAnodeFrontAxisY.commandConfiguration.camIn.syncProfileReference := 1;
   cmMendrelAnodeFrontAxisY.commandConfiguration.camIn.masterStartDistance := 0.0;
   cmMendrelAnodeFrontAxisY.commandConfiguration.camIn.velocity := -1.0;
   cmMendrelAnodeFrontAxisY.commandConfiguration.camIn.acceleration := -1.0;
   cmMendrelAnodeFrontAxisY.commandConfiguration.camIn.deceleration := -1.0;
   cmMendrelAnodeFrontAxisY.commandConfiguration.camIn.jerk := -1.0;
   cmMendrelAnodeFrontAxisY.commandConfiguration.camIn.applicationMode := 0;
   cmMendrelAnodeFrontAxisY.commandConfiguration.camIn.syncDirection := 1;
   cmMendrelAnodeFrontAxisY.commandConfiguration.gearOutCamOut.slavePosition := 0.0;
   cmMendrelAnodeFrontAxisY.commandConfiguration.gearOutCamOut.syncProfileReference := 1;
   cmMendrelAnodeFrontAxisY.commandConfiguration.gearOutCamOut.masterStopDistance := 0.0;
   cmMendrelAnodeFrontAxisY.commandConfiguration.gearOutCamOut.deceleration := -1.0;
   cmMendrelAnodeFrontAxisY.commandConfiguration.gearOutCamOut.jerk := -1.0;
   cmMendrelAnodeFrontAxisY.commandConfiguration.gearOutCamOut.syncOutDirection := 3;
   cmMendrelAnodeFrontAxisY.commandConfiguration.gearOutCamOut.gearOutCamOutMode := -1;
   cmMendrelAnodeFrontAxisY.commandConfiguration.phasing.phaseShift := 0.0;
   cmMendrelAnodeFrontAxisY.commandConfiguration.phasing.velocity := -1.0;
   cmMendrelAnodeFrontAxisY.commandConfiguration.phasing.acceleration := -1.0;
   cmMendrelAnodeFrontAxisY.commandConfiguration.phasing.deceleration := -1.0;
   cmMendrelAnodeFrontAxisY.commandConfiguration.phasing.jerk := -1.0;
   cmMendrelAnodeFrontAxisY.commandConfiguration.phasing.profileReference := 0;
   cmMendrelAnodeFrontAxisY.commandConfiguration.phasing.phasingDistance := 0.0;
   cmMendrelAnodeFrontAxisY.commandConfiguration.phasing.startPosition := 0.0;
   cmMendrelAnodeFrontAxisY.commandConfiguration.phasing.direction := 3;
   cmMendrelAnodeFrontAxisY.commandConfiguration.phasing.phaseAbsolute := TRUE;
   cmMendrelAnodeFrontAxisY.commandConfiguration.phasing.phaseShiftChangeOnTheFly := FALSE;
   cmMendrelAnodeFrontAxisY.commandConfiguration.offset.offset := 0.0;
   cmMendrelAnodeFrontAxisY.commandConfiguration.offset.profileReference := 1;
   cmMendrelAnodeFrontAxisY.commandConfiguration.offset.offsetDistance := 0.0;
   cmMendrelAnodeFrontAxisY.commandConfiguration.offset.startPosition := 0.0;
   cmMendrelAnodeFrontAxisY.commandConfiguration.offset.direction := 3;
   cmMendrelAnodeFrontAxisY.commandConfiguration.offset.offsetAbsolute := TRUE;
   cmMendrelAnodeFrontAxisY.commandConfiguration.offset.offsetChangeOnTheFly := FALSE;
   cmMendrelAnodeFrontAxisY.commands.enableAxis := FALSE;
   cmMendrelAnodeFrontAxisY.commands.resetAxis := FALSE;
   cmMendrelAnodeFrontAxisY.commands.openBrake := FALSE;
   cmMendrelAnodeFrontAxisY.commands.jogForward := FALSE;
   cmMendrelAnodeFrontAxisY.commands.jogBackward := FALSE;
   cmMendrelAnodeFrontAxisY.commands.moveVelocity := FALSE;
   cmMendrelAnodeFrontAxisY.commands.stop := FALSE;
   cmMendrelAnodeFrontAxisY.commands.fastStop := FALSE;
   cmMendrelAnodeFrontAxisY.commands.torqueLimiting := FALSE;
   cmMendrelAnodeFrontAxisY.commands.homing := FALSE;
   cmMendrelAnodeFrontAxisY.commands.posRelative := FALSE;
   cmMendrelAnodeFrontAxisY.commands.posAbsolute := FALSE;
   cmMendrelAnodeFrontAxisY.commands.posSuperimposed := FALSE;
   cmMendrelAnodeFrontAxisY.commands.haltSuperimposed := FALSE;
   cmMendrelAnodeFrontAxisY.commands.selectSetPosition := -1;
   cmMendrelAnodeFrontAxisY.commands.reset := FALSE;
   cmMendrelAnodeFrontAxisY.monitoring.valid := FALSE;
   cmMendrelAnodeFrontAxisY.monitoring.busy := TRUE;
   cmMendrelAnodeFrontAxisY.monitoring.error := TRUE;
   cmMendrelAnodeFrontAxisY.monitoring.status := 16#8600;
   cmMendrelAnodeFrontAxisY.monitoring.subfunctionStatus := 16#8001;
   cmMendrelAnodeFrontAxisY.monitoring.axisEnabled := FALSE;
   cmMendrelAnodeFrontAxisY.monitoring.resetActive := FALSE;
   cmMendrelAnodeFrontAxisY.monitoring.inVelocity := FALSE;
   cmMendrelAnodeFrontAxisY.monitoring.inLimitation := FALSE;
   cmMendrelAnodeFrontAxisY.monitoring.inClamping := FALSE;
   cmMendrelAnodeFrontAxisY.monitoring.startSync := FALSE;
   cmMendrelAnodeFrontAxisY.monitoring.inSync := FALSE;
   cmMendrelAnodeFrontAxisY.monitoring.inSimulation := FALSE;
   cmMendrelAnodeFrontAxisY.monitoring.jogSelected := FALSE;
   cmMendrelAnodeFrontAxisY.monitoring.moveVelocitySelected := FALSE;
   cmMendrelAnodeFrontAxisY.monitoring.stopSelected := FALSE;
   cmMendrelAnodeFrontAxisY.monitoring.fastStopSelected := FALSE;
   cmMendrelAnodeFrontAxisY.monitoring.torqueLimitingSelected := FALSE;
   cmMendrelAnodeFrontAxisY.monitoring.homingSelected := FALSE;
   cmMendrelAnodeFrontAxisY.monitoring.posRelativeSelected := FALSE;
   cmMendrelAnodeFrontAxisY.monitoring.posAbsoluteSelected := FALSE;
   cmMendrelAnodeFrontAxisY.monitoring.posSuperimposedSelected := FALSE;
   cmMendrelAnodeFrontAxisY.monitoring.haltSuperimposedSelected := FALSE;
   cmMendrelAnodeFrontAxisY.monitoring.commandBusy := FALSE;
   cmMendrelAnodeFrontAxisY.monitoring.commandDone := FALSE;
   cmMendrelAnodeFrontAxisY.monitoring.commandAborted := FALSE;
   cmMendrelAnodeFrontAxisY.monitoring.homingCommandBusy := FALSE;
   cmMendrelAnodeFrontAxisY.monitoring.homingCommandDone := FALSE;
   cmMendrelAnodeFrontAxisY.monitoring.homingCommandAborted := FALSE;
   cmMendrelAnodeFrontAxisY.monitoring.superimposedBusy := FALSE;
   cmMendrelAnodeFrontAxisY.monitoring.superimposedDone := FALSE;
   cmMendrelAnodeFrontAxisY.monitoring.superimposedAborted := FALSE;
   cmMendrelAnodeFrontAxisY.monitoring.actualPosition := 43.33;
   cmMendrelAnodeFrontAxisY.monitoring.actualSpeed := 0.0;
   cmMendrelAnodeFrontAxisY.monitoring.speedUnit := 1062;
   cmMendrelAnodeFrontAxisY.monitoring.positionUnit := 1013;
   cmMendrelAnodeFrontAxisY.monitoring.axisType := 1;
   cmMendrelAnodeFrontAxisY.monitoring.interlockGeneralOut := TRUE;
   cmMendrelAnodeFrontAxisY.monitoring.interlockJogForwardOut := TRUE;
   cmMendrelAnodeFrontAxisY.monitoring.interlockJogBackwardOut := TRUE;
   cmMendrelAnodeFrontAxisZ.commandConfiguration.generalSettings.stopOnError := TRUE;
   cmMendrelAnodeFrontAxisZ.commandConfiguration.generalSettings.resetWithRestart := FALSE;
   cmMendrelAnodeFrontAxisZ.commandConfiguration.generalSettings.abortWaitingSyncCmd := TRUE;
   cmMendrelAnodeFrontAxisZ.commandConfiguration.power.startMode := 1;
   cmMendrelAnodeFrontAxisZ.commandConfiguration.power.stopMode := 0;
   cmMendrelAnodeFrontAxisZ.commandConfiguration.power.syncMotionSimulation := FALSE;
   cmMendrelAnodeFrontAxisZ.commandConfiguration.power.syncMotionSimulationExtendedMode := -1;
   cmMendrelAnodeFrontAxisZ.commandConfiguration.jog.velocity := 5.0;
   cmMendrelAnodeFrontAxisZ.commandConfiguration.jog.acceleration := 50.0;
   cmMendrelAnodeFrontAxisZ.commandConfiguration.jog.deceleration := 50.0;
   cmMendrelAnodeFrontAxisZ.commandConfiguration.jog.jerk := -1.0;
   cmMendrelAnodeFrontAxisZ.commandConfiguration.jog.positionControlled := TRUE;
   cmMendrelAnodeFrontAxisZ.commandConfiguration.jog.increment := 0.0;
   cmMendrelAnodeFrontAxisZ.commandConfiguration.jog.mode := 0;
   cmMendrelAnodeFrontAxisZ.commandConfiguration.moveVelocity.velocity := 0.0;
   cmMendrelAnodeFrontAxisZ.commandConfiguration.moveVelocity.acceleration := -1.0;
   cmMendrelAnodeFrontAxisZ.commandConfiguration.moveVelocity.deceleration := -1.0;
   cmMendrelAnodeFrontAxisZ.commandConfiguration.moveVelocity.jerk := -1.0;
   cmMendrelAnodeFrontAxisZ.commandConfiguration.moveVelocity.direction := 0;
   cmMendrelAnodeFrontAxisZ.commandConfiguration.moveVelocity.positionControlled := TRUE;
   cmMendrelAnodeFrontAxisZ.commandConfiguration.moveVelocity.velocityChangeOnTheFly := FALSE;
   cmMendrelAnodeFrontAxisZ.commandConfiguration.stop.deceleration := -1.0;
   cmMendrelAnodeFrontAxisZ.commandConfiguration.stop.jerk := -1.0;
   cmMendrelAnodeFrontAxisZ.commandConfiguration.stop.abortAcceleration := FALSE;
   cmMendrelAnodeFrontAxisZ.commandConfiguration.fastStop.deceleration := -1.0;
   cmMendrelAnodeFrontAxisZ.commandConfiguration.fastStop.jerk := -1.0;
   cmMendrelAnodeFrontAxisZ.commandConfiguration.fastStop.abortAcceleration := FALSE;
   cmMendrelAnodeFrontAxisZ.commandConfiguration.fastStop.replaceStopPossible := FALSE;
   cmMendrelAnodeFrontAxisZ.commandConfiguration.torqueLimiting.limit := -1.0;
   cmMendrelAnodeFrontAxisZ.commandConfiguration.torqueLimiting.mode := 0;
   cmMendrelAnodeFrontAxisZ.commandConfiguration.homing.position := 0.0;
   cmMendrelAnodeFrontAxisZ.commandConfiguration.homing.mode := 0;
   cmMendrelAnodeFrontAxisZ.commandConfiguration.homing.sensor := 0;
   cmMendrelAnodeFrontAxisZ.commandConfiguration.homing.extendedMode := -1;
   cmMendrelAnodeFrontAxisZ.commandConfiguration.homing.extendedModeTorqueLimit := 0.0;
   cmMendrelAnodeFrontAxisZ.commandConfiguration.homing.extendedModeTargetPosition := 0.0;
   cmMendrelAnodeFrontAxisZ.commandConfiguration.posRelative.distance := 0.0;
   cmMendrelAnodeFrontAxisZ.commandConfiguration.posRelative.velocity := -1.0;
   cmMendrelAnodeFrontAxisZ.commandConfiguration.posRelative.acceleration := -1.0;
   cmMendrelAnodeFrontAxisZ.commandConfiguration.posRelative.deceleration := -1.0;
   cmMendrelAnodeFrontAxisZ.commandConfiguration.posRelative.jerk := -1.0;
   cmMendrelAnodeFrontAxisZ.commandConfiguration.posRelative.direction := 0;
   cmMendrelAnodeFrontAxisZ.commandConfiguration.posAbsolute.position := -2.8;
   cmMendrelAnodeFrontAxisZ.commandConfiguration.posAbsolute.velocity := 30.0;
   cmMendrelAnodeFrontAxisZ.commandConfiguration.posAbsolute.acceleration := 30.0;
   cmMendrelAnodeFrontAxisZ.commandConfiguration.posAbsolute.deceleration := 30.0;
   cmMendrelAnodeFrontAxisZ.commandConfiguration.posAbsolute.jerk := -1.0;
   cmMendrelAnodeFrontAxisZ.commandConfiguration.posAbsolute.direction := 1;
   cmMendrelAnodeFrontAxisZ.commandConfiguration.posAbsolute.positionChangeOnTheFly := FALSE;
   cmMendrelAnodeFrontAxisZ.commandConfiguration.posAbsolute.velocityChangeOnTheFly := FALSE;
   cmMendrelAnodeFrontAxisZ.commandConfiguration.posSuperimposed.distance := 0.0;
   cmMendrelAnodeFrontAxisZ.commandConfiguration.posSuperimposed.velocityDiff := -1.0;
   cmMendrelAnodeFrontAxisZ.commandConfiguration.posSuperimposed.acceleration := -1.0;
   cmMendrelAnodeFrontAxisZ.commandConfiguration.posSuperimposed.deceleration := -1.0;
   cmMendrelAnodeFrontAxisZ.commandConfiguration.posSuperimposed.jerk := -1.0;
   cmMendrelAnodeFrontAxisZ.commandConfiguration.posSuperimposed.direction := 0;
   cmMendrelAnodeFrontAxisZ.commandConfiguration.haltSuperimposed.deceleration := -1.0;
   cmMendrelAnodeFrontAxisZ.commandConfiguration.haltSuperimposed.jerk := -1.0;
   cmMendrelAnodeFrontAxisZ.commandConfiguration.haltSuperimposed.abortAcceleration := FALSE;
   cmMendrelAnodeFrontAxisZ.commandConfiguration.gearInRelative.ratioNumerator := 1;
   cmMendrelAnodeFrontAxisZ.commandConfiguration.gearInRelative.ratioDenominator := 1;
   cmMendrelAnodeFrontAxisZ.commandConfiguration.gearInRelative.acceleration := -1.0;
   cmMendrelAnodeFrontAxisZ.commandConfiguration.gearInRelative.deceleration := -1.0;
   cmMendrelAnodeFrontAxisZ.commandConfiguration.gearInRelative.jerk := -1.0;
   cmMendrelAnodeFrontAxisZ.commandConfiguration.gearInRelative.ratioChangeOnTheFly := FALSE;
   cmMendrelAnodeFrontAxisZ.commandConfiguration.gearInAbsolute.ratioNumerator := 1;
   cmMendrelAnodeFrontAxisZ.commandConfiguration.gearInAbsolute.ratioDenominator := 1;
   cmMendrelAnodeFrontAxisZ.commandConfiguration.gearInAbsolute.masterSyncPosition := 0.0;
   cmMendrelAnodeFrontAxisZ.commandConfiguration.gearInAbsolute.slaveSyncPosition := 0.0;
   cmMendrelAnodeFrontAxisZ.commandConfiguration.gearInAbsolute.syncProfileReference := 1;
   cmMendrelAnodeFrontAxisZ.commandConfiguration.gearInAbsolute.masterStartDistance := 0.0;
   cmMendrelAnodeFrontAxisZ.commandConfiguration.gearInAbsolute.velocity := -1.0;
   cmMendrelAnodeFrontAxisZ.commandConfiguration.gearInAbsolute.acceleration := -1.0;
   cmMendrelAnodeFrontAxisZ.commandConfiguration.gearInAbsolute.deceleration := -1.0;
   cmMendrelAnodeFrontAxisZ.commandConfiguration.gearInAbsolute.jerk := -1.0;
   cmMendrelAnodeFrontAxisZ.commandConfiguration.gearInAbsolute.syncDirection := 1;
   cmMendrelAnodeFrontAxisZ.commandConfiguration.gearInAbsolute.ratioChangeOnTheFly := FALSE;
   cmMendrelAnodeFrontAxisZ.commandConfiguration.gearInVelocity.continuousUpdate := FALSE;
   cmMendrelAnodeFrontAxisZ.commandConfiguration.gearInVelocity.ratioNumerator := 1;
   cmMendrelAnodeFrontAxisZ.commandConfiguration.gearInVelocity.ratioDenominator := 1;
   cmMendrelAnodeFrontAxisZ.commandConfiguration.gearInVelocity.acceleration := -1.0;
   cmMendrelAnodeFrontAxisZ.commandConfiguration.gearInVelocity.deceleration := -1.0;
   cmMendrelAnodeFrontAxisZ.commandConfiguration.gearInVelocity.jerk := -1.0;
   cmMendrelAnodeFrontAxisZ.commandConfiguration.gearInVelocity.positionControlled := FALSE;
   cmMendrelAnodeFrontAxisZ.commandConfiguration.camIn.masterOffset := 0.0;
   cmMendrelAnodeFrontAxisZ.commandConfiguration.camIn.slaveOffset := 0.0;
   cmMendrelAnodeFrontAxisZ.commandConfiguration.camIn.masterScaling := 1.0;
   cmMendrelAnodeFrontAxisZ.commandConfiguration.camIn.slaveScaling := 1.0;
   cmMendrelAnodeFrontAxisZ.commandConfiguration.camIn.masterSyncPosition := 0.0;
   cmMendrelAnodeFrontAxisZ.commandConfiguration.camIn.syncProfileReference := 1;
   cmMendrelAnodeFrontAxisZ.commandConfiguration.camIn.masterStartDistance := 0.0;
   cmMendrelAnodeFrontAxisZ.commandConfiguration.camIn.velocity := -1.0;
   cmMendrelAnodeFrontAxisZ.commandConfiguration.camIn.acceleration := -1.0;
   cmMendrelAnodeFrontAxisZ.commandConfiguration.camIn.deceleration := -1.0;
   cmMendrelAnodeFrontAxisZ.commandConfiguration.camIn.jerk := -1.0;
   cmMendrelAnodeFrontAxisZ.commandConfiguration.camIn.applicationMode := 0;
   cmMendrelAnodeFrontAxisZ.commandConfiguration.camIn.syncDirection := 1;
   cmMendrelAnodeFrontAxisZ.commandConfiguration.gearOutCamOut.slavePosition := 0.0;
   cmMendrelAnodeFrontAxisZ.commandConfiguration.gearOutCamOut.syncProfileReference := 1;
   cmMendrelAnodeFrontAxisZ.commandConfiguration.gearOutCamOut.masterStopDistance := 0.0;
   cmMendrelAnodeFrontAxisZ.commandConfiguration.gearOutCamOut.deceleration := -1.0;
   cmMendrelAnodeFrontAxisZ.commandConfiguration.gearOutCamOut.jerk := -1.0;
   cmMendrelAnodeFrontAxisZ.commandConfiguration.gearOutCamOut.syncOutDirection := 3;
   cmMendrelAnodeFrontAxisZ.commandConfiguration.gearOutCamOut.gearOutCamOutMode := -1;
   cmMendrelAnodeFrontAxisZ.commandConfiguration.phasing.phaseShift := 0.0;
   cmMendrelAnodeFrontAxisZ.commandConfiguration.phasing.velocity := -1.0;
   cmMendrelAnodeFrontAxisZ.commandConfiguration.phasing.acceleration := -1.0;
   cmMendrelAnodeFrontAxisZ.commandConfiguration.phasing.deceleration := -1.0;
   cmMendrelAnodeFrontAxisZ.commandConfiguration.phasing.jerk := -1.0;
   cmMendrelAnodeFrontAxisZ.commandConfiguration.phasing.profileReference := 0;
   cmMendrelAnodeFrontAxisZ.commandConfiguration.phasing.phasingDistance := 0.0;
   cmMendrelAnodeFrontAxisZ.commandConfiguration.phasing.startPosition := 0.0;
   cmMendrelAnodeFrontAxisZ.commandConfiguration.phasing.direction := 3;
   cmMendrelAnodeFrontAxisZ.commandConfiguration.phasing.phaseAbsolute := TRUE;
   cmMendrelAnodeFrontAxisZ.commandConfiguration.phasing.phaseShiftChangeOnTheFly := FALSE;
   cmMendrelAnodeFrontAxisZ.commandConfiguration.offset.offset := 0.0;
   cmMendrelAnodeFrontAxisZ.commandConfiguration.offset.profileReference := 1;
   cmMendrelAnodeFrontAxisZ.commandConfiguration.offset.offsetDistance := 0.0;
   cmMendrelAnodeFrontAxisZ.commandConfiguration.offset.startPosition := 0.0;
   cmMendrelAnodeFrontAxisZ.commandConfiguration.offset.direction := 3;
   cmMendrelAnodeFrontAxisZ.commandConfiguration.offset.offsetAbsolute := TRUE;
   cmMendrelAnodeFrontAxisZ.commandConfiguration.offset.offsetChangeOnTheFly := FALSE;
   cmMendrelAnodeFrontAxisZ.commands.enableAxis := FALSE;
   cmMendrelAnodeFrontAxisZ.commands.resetAxis := FALSE;
   cmMendrelAnodeFrontAxisZ.commands.openBrake := FALSE;
   cmMendrelAnodeFrontAxisZ.commands.jogForward := FALSE;
   cmMendrelAnodeFrontAxisZ.commands.jogBackward := FALSE;
   cmMendrelAnodeFrontAxisZ.commands.moveVelocity := FALSE;
   cmMendrelAnodeFrontAxisZ.commands.stop := FALSE;
   cmMendrelAnodeFrontAxisZ.commands.fastStop := FALSE;
   cmMendrelAnodeFrontAxisZ.commands.torqueLimiting := FALSE;
   cmMendrelAnodeFrontAxisZ.commands.homing := FALSE;
   cmMendrelAnodeFrontAxisZ.commands.posRelative := FALSE;
   cmMendrelAnodeFrontAxisZ.commands.posAbsolute := FALSE;
   cmMendrelAnodeFrontAxisZ.commands.posSuperimposed := FALSE;
   cmMendrelAnodeFrontAxisZ.commands.haltSuperimposed := FALSE;
   cmMendrelAnodeFrontAxisZ.commands.selectSetPosition := -1;
   cmMendrelAnodeFrontAxisZ.commands.reset := FALSE;
   cmMendrelAnodeFrontAxisZ.monitoring.valid := FALSE;
   cmMendrelAnodeFrontAxisZ.monitoring.busy := TRUE;
   cmMendrelAnodeFrontAxisZ.monitoring.error := TRUE;
   cmMendrelAnodeFrontAxisZ.monitoring.status := 16#8600;
   cmMendrelAnodeFrontAxisZ.monitoring.subfunctionStatus := 16#8001;
   cmMendrelAnodeFrontAxisZ.monitoring.axisEnabled := FALSE;
   cmMendrelAnodeFrontAxisZ.monitoring.resetActive := FALSE;
   cmMendrelAnodeFrontAxisZ.monitoring.inVelocity := FALSE;
   cmMendrelAnodeFrontAxisZ.monitoring.inLimitation := FALSE;
   cmMendrelAnodeFrontAxisZ.monitoring.inClamping := FALSE;
   cmMendrelAnodeFrontAxisZ.monitoring.startSync := FALSE;
   cmMendrelAnodeFrontAxisZ.monitoring.inSync := FALSE;
   cmMendrelAnodeFrontAxisZ.monitoring.inSimulation := FALSE;
   cmMendrelAnodeFrontAxisZ.monitoring.jogSelected := FALSE;
   cmMendrelAnodeFrontAxisZ.monitoring.moveVelocitySelected := FALSE;
   cmMendrelAnodeFrontAxisZ.monitoring.stopSelected := FALSE;
   cmMendrelAnodeFrontAxisZ.monitoring.fastStopSelected := FALSE;
   cmMendrelAnodeFrontAxisZ.monitoring.torqueLimitingSelected := FALSE;
   cmMendrelAnodeFrontAxisZ.monitoring.homingSelected := FALSE;
   cmMendrelAnodeFrontAxisZ.monitoring.posRelativeSelected := FALSE;
   cmMendrelAnodeFrontAxisZ.monitoring.posAbsoluteSelected := FALSE;
   cmMendrelAnodeFrontAxisZ.monitoring.posSuperimposedSelected := FALSE;
   cmMendrelAnodeFrontAxisZ.monitoring.haltSuperimposedSelected := FALSE;
   cmMendrelAnodeFrontAxisZ.monitoring.commandBusy := FALSE;
   cmMendrelAnodeFrontAxisZ.monitoring.commandDone := FALSE;
   cmMendrelAnodeFrontAxisZ.monitoring.commandAborted := FALSE;
   cmMendrelAnodeFrontAxisZ.monitoring.homingCommandBusy := FALSE;
   cmMendrelAnodeFrontAxisZ.monitoring.homingCommandDone := FALSE;
   cmMendrelAnodeFrontAxisZ.monitoring.homingCommandAborted := FALSE;
   cmMendrelAnodeFrontAxisZ.monitoring.superimposedBusy := FALSE;
   cmMendrelAnodeFrontAxisZ.monitoring.superimposedDone := FALSE;
   cmMendrelAnodeFrontAxisZ.monitoring.superimposedAborted := FALSE;
   cmMendrelAnodeFrontAxisZ.monitoring.actualPosition := 20.88;
   cmMendrelAnodeFrontAxisZ.monitoring.actualSpeed := 0.0;
   cmMendrelAnodeFrontAxisZ.monitoring.speedUnit := 1062;
   cmMendrelAnodeFrontAxisZ.monitoring.positionUnit := 1013;
   cmMendrelAnodeFrontAxisZ.monitoring.axisType := 1;
   cmMendrelAnodeFrontAxisZ.monitoring.interlockGeneralOut := TRUE;
   cmMendrelAnodeFrontAxisZ.monitoring.interlockJogForwardOut := TRUE;
   cmMendrelAnodeFrontAxisZ.monitoring.interlockJogBackwardOut := TRUE;
   cmMendrelAnodeRearAxisY.commandConfiguration.generalSettings.stopOnError := TRUE;
   cmMendrelAnodeRearAxisY.commandConfiguration.generalSettings.resetWithRestart := FALSE;
   cmMendrelAnodeRearAxisY.commandConfiguration.generalSettings.abortWaitingSyncCmd := TRUE;
   cmMendrelAnodeRearAxisY.commandConfiguration.power.startMode := 1;
   cmMendrelAnodeRearAxisY.commandConfiguration.power.stopMode := 0;
   cmMendrelAnodeRearAxisY.commandConfiguration.power.syncMotionSimulation := FALSE;
   cmMendrelAnodeRearAxisY.commandConfiguration.power.syncMotionSimulationExtendedMode := -1;
   cmMendrelAnodeRearAxisY.commandConfiguration.jog.velocity := 0.0;
   cmMendrelAnodeRearAxisY.commandConfiguration.jog.acceleration := -1.0;
   cmMendrelAnodeRearAxisY.commandConfiguration.jog.deceleration := -1.0;
   cmMendrelAnodeRearAxisY.commandConfiguration.jog.jerk := -1.0;
   cmMendrelAnodeRearAxisY.commandConfiguration.jog.positionControlled := TRUE;
   cmMendrelAnodeRearAxisY.commandConfiguration.jog.increment := 0.0;
   cmMendrelAnodeRearAxisY.commandConfiguration.jog.mode := 0;
   cmMendrelAnodeRearAxisY.commandConfiguration.moveVelocity.velocity := 0.0;
   cmMendrelAnodeRearAxisY.commandConfiguration.moveVelocity.acceleration := -1.0;
   cmMendrelAnodeRearAxisY.commandConfiguration.moveVelocity.deceleration := -1.0;
   cmMendrelAnodeRearAxisY.commandConfiguration.moveVelocity.jerk := -1.0;
   cmMendrelAnodeRearAxisY.commandConfiguration.moveVelocity.direction := 0;
   cmMendrelAnodeRearAxisY.commandConfiguration.moveVelocity.positionControlled := TRUE;
   cmMendrelAnodeRearAxisY.commandConfiguration.moveVelocity.velocityChangeOnTheFly := FALSE;
   cmMendrelAnodeRearAxisY.commandConfiguration.stop.deceleration := -1.0;
   cmMendrelAnodeRearAxisY.commandConfiguration.stop.jerk := -1.0;
   cmMendrelAnodeRearAxisY.commandConfiguration.stop.abortAcceleration := FALSE;
   cmMendrelAnodeRearAxisY.commandConfiguration.fastStop.deceleration := -1.0;
   cmMendrelAnodeRearAxisY.commandConfiguration.fastStop.jerk := -1.0;
   cmMendrelAnodeRearAxisY.commandConfiguration.fastStop.abortAcceleration := FALSE;
   cmMendrelAnodeRearAxisY.commandConfiguration.fastStop.replaceStopPossible := FALSE;
   cmMendrelAnodeRearAxisY.commandConfiguration.torqueLimiting.limit := -1.0;
   cmMendrelAnodeRearAxisY.commandConfiguration.torqueLimiting.mode := 0;
   cmMendrelAnodeRearAxisY.commandConfiguration.homing.position := 0.0;
   cmMendrelAnodeRearAxisY.commandConfiguration.homing.mode := 0;
   cmMendrelAnodeRearAxisY.commandConfiguration.homing.sensor := 0;
   cmMendrelAnodeRearAxisY.commandConfiguration.homing.extendedMode := -1;
   cmMendrelAnodeRearAxisY.commandConfiguration.homing.extendedModeTorqueLimit := 0.0;
   cmMendrelAnodeRearAxisY.commandConfiguration.homing.extendedModeTargetPosition := 0.0;
   cmMendrelAnodeRearAxisY.commandConfiguration.posRelative.distance := 0.0;
   cmMendrelAnodeRearAxisY.commandConfiguration.posRelative.velocity := -1.0;
   cmMendrelAnodeRearAxisY.commandConfiguration.posRelative.acceleration := -1.0;
   cmMendrelAnodeRearAxisY.commandConfiguration.posRelative.deceleration := -1.0;
   cmMendrelAnodeRearAxisY.commandConfiguration.posRelative.jerk := -1.0;
   cmMendrelAnodeRearAxisY.commandConfiguration.posRelative.direction := 0;
   cmMendrelAnodeRearAxisY.commandConfiguration.posAbsolute.position := 0.0;
   cmMendrelAnodeRearAxisY.commandConfiguration.posAbsolute.velocity := -1.0;
   cmMendrelAnodeRearAxisY.commandConfiguration.posAbsolute.acceleration := -1.0;
   cmMendrelAnodeRearAxisY.commandConfiguration.posAbsolute.deceleration := -1.0;
   cmMendrelAnodeRearAxisY.commandConfiguration.posAbsolute.jerk := -1.0;
   cmMendrelAnodeRearAxisY.commandConfiguration.posAbsolute.direction := 1;
   cmMendrelAnodeRearAxisY.commandConfiguration.posAbsolute.positionChangeOnTheFly := FALSE;
   cmMendrelAnodeRearAxisY.commandConfiguration.posAbsolute.velocityChangeOnTheFly := FALSE;
   cmMendrelAnodeRearAxisY.commandConfiguration.posSuperimposed.distance := 0.0;
   cmMendrelAnodeRearAxisY.commandConfiguration.posSuperimposed.velocityDiff := -1.0;
   cmMendrelAnodeRearAxisY.commandConfiguration.posSuperimposed.acceleration := -1.0;
   cmMendrelAnodeRearAxisY.commandConfiguration.posSuperimposed.deceleration := -1.0;
   cmMendrelAnodeRearAxisY.commandConfiguration.posSuperimposed.jerk := -1.0;
   cmMendrelAnodeRearAxisY.commandConfiguration.posSuperimposed.direction := 0;
   cmMendrelAnodeRearAxisY.commandConfiguration.haltSuperimposed.deceleration := -1.0;
   cmMendrelAnodeRearAxisY.commandConfiguration.haltSuperimposed.jerk := -1.0;
   cmMendrelAnodeRearAxisY.commandConfiguration.haltSuperimposed.abortAcceleration := FALSE;
   cmMendrelAnodeRearAxisY.commandConfiguration.gearInRelative.ratioNumerator := 1;
   cmMendrelAnodeRearAxisY.commandConfiguration.gearInRelative.ratioDenominator := 1;
   cmMendrelAnodeRearAxisY.commandConfiguration.gearInRelative.acceleration := -1.0;
   cmMendrelAnodeRearAxisY.commandConfiguration.gearInRelative.deceleration := -1.0;
   cmMendrelAnodeRearAxisY.commandConfiguration.gearInRelative.jerk := -1.0;
   cmMendrelAnodeRearAxisY.commandConfiguration.gearInRelative.ratioChangeOnTheFly := FALSE;
   cmMendrelAnodeRearAxisY.commandConfiguration.gearInAbsolute.ratioNumerator := 1;
   cmMendrelAnodeRearAxisY.commandConfiguration.gearInAbsolute.ratioDenominator := 1;
   cmMendrelAnodeRearAxisY.commandConfiguration.gearInAbsolute.masterSyncPosition := 0.0;
   cmMendrelAnodeRearAxisY.commandConfiguration.gearInAbsolute.slaveSyncPosition := 0.0;
   cmMendrelAnodeRearAxisY.commandConfiguration.gearInAbsolute.syncProfileReference := 1;
   cmMendrelAnodeRearAxisY.commandConfiguration.gearInAbsolute.masterStartDistance := 0.0;
   cmMendrelAnodeRearAxisY.commandConfiguration.gearInAbsolute.velocity := -1.0;
   cmMendrelAnodeRearAxisY.commandConfiguration.gearInAbsolute.acceleration := -1.0;
   cmMendrelAnodeRearAxisY.commandConfiguration.gearInAbsolute.deceleration := -1.0;
   cmMendrelAnodeRearAxisY.commandConfiguration.gearInAbsolute.jerk := -1.0;
   cmMendrelAnodeRearAxisY.commandConfiguration.gearInAbsolute.syncDirection := 1;
   cmMendrelAnodeRearAxisY.commandConfiguration.gearInAbsolute.ratioChangeOnTheFly := FALSE;
   cmMendrelAnodeRearAxisY.commandConfiguration.gearInVelocity.continuousUpdate := FALSE;
   cmMendrelAnodeRearAxisY.commandConfiguration.gearInVelocity.ratioNumerator := 1;
   cmMendrelAnodeRearAxisY.commandConfiguration.gearInVelocity.ratioDenominator := 1;
   cmMendrelAnodeRearAxisY.commandConfiguration.gearInVelocity.acceleration := -1.0;
   cmMendrelAnodeRearAxisY.commandConfiguration.gearInVelocity.deceleration := -1.0;
   cmMendrelAnodeRearAxisY.commandConfiguration.gearInVelocity.jerk := -1.0;
   cmMendrelAnodeRearAxisY.commandConfiguration.gearInVelocity.positionControlled := FALSE;
   cmMendrelAnodeRearAxisY.commandConfiguration.camIn.masterOffset := 0.0;
   cmMendrelAnodeRearAxisY.commandConfiguration.camIn.slaveOffset := 0.0;
   cmMendrelAnodeRearAxisY.commandConfiguration.camIn.masterScaling := 1.0;
   cmMendrelAnodeRearAxisY.commandConfiguration.camIn.slaveScaling := 1.0;
   cmMendrelAnodeRearAxisY.commandConfiguration.camIn.masterSyncPosition := 0.0;
   cmMendrelAnodeRearAxisY.commandConfiguration.camIn.syncProfileReference := 1;
   cmMendrelAnodeRearAxisY.commandConfiguration.camIn.masterStartDistance := 0.0;
   cmMendrelAnodeRearAxisY.commandConfiguration.camIn.velocity := -1.0;
   cmMendrelAnodeRearAxisY.commandConfiguration.camIn.acceleration := -1.0;
   cmMendrelAnodeRearAxisY.commandConfiguration.camIn.deceleration := -1.0;
   cmMendrelAnodeRearAxisY.commandConfiguration.camIn.jerk := -1.0;
   cmMendrelAnodeRearAxisY.commandConfiguration.camIn.applicationMode := 0;
   cmMendrelAnodeRearAxisY.commandConfiguration.camIn.syncDirection := 1;
   cmMendrelAnodeRearAxisY.commandConfiguration.gearOutCamOut.slavePosition := 0.0;
   cmMendrelAnodeRearAxisY.commandConfiguration.gearOutCamOut.syncProfileReference := 1;
   cmMendrelAnodeRearAxisY.commandConfiguration.gearOutCamOut.masterStopDistance := 0.0;
   cmMendrelAnodeRearAxisY.commandConfiguration.gearOutCamOut.deceleration := -1.0;
   cmMendrelAnodeRearAxisY.commandConfiguration.gearOutCamOut.jerk := -1.0;
   cmMendrelAnodeRearAxisY.commandConfiguration.gearOutCamOut.syncOutDirection := 3;
   cmMendrelAnodeRearAxisY.commandConfiguration.gearOutCamOut.gearOutCamOutMode := -1;
   cmMendrelAnodeRearAxisY.commandConfiguration.phasing.phaseShift := 0.0;
   cmMendrelAnodeRearAxisY.commandConfiguration.phasing.velocity := -1.0;
   cmMendrelAnodeRearAxisY.commandConfiguration.phasing.acceleration := -1.0;
   cmMendrelAnodeRearAxisY.commandConfiguration.phasing.deceleration := -1.0;
   cmMendrelAnodeRearAxisY.commandConfiguration.phasing.jerk := -1.0;
   cmMendrelAnodeRearAxisY.commandConfiguration.phasing.profileReference := 0;
   cmMendrelAnodeRearAxisY.commandConfiguration.phasing.phasingDistance := 0.0;
   cmMendrelAnodeRearAxisY.commandConfiguration.phasing.startPosition := 0.0;
   cmMendrelAnodeRearAxisY.commandConfiguration.phasing.direction := 3;
   cmMendrelAnodeRearAxisY.commandConfiguration.phasing.phaseAbsolute := TRUE;
   cmMendrelAnodeRearAxisY.commandConfiguration.phasing.phaseShiftChangeOnTheFly := FALSE;
   cmMendrelAnodeRearAxisY.commandConfiguration.offset.offset := 0.0;
   cmMendrelAnodeRearAxisY.commandConfiguration.offset.profileReference := 1;
   cmMendrelAnodeRearAxisY.commandConfiguration.offset.offsetDistance := 0.0;
   cmMendrelAnodeRearAxisY.commandConfiguration.offset.startPosition := 0.0;
   cmMendrelAnodeRearAxisY.commandConfiguration.offset.direction := 3;
   cmMendrelAnodeRearAxisY.commandConfiguration.offset.offsetAbsolute := TRUE;
   cmMendrelAnodeRearAxisY.commandConfiguration.offset.offsetChangeOnTheFly := FALSE;
   cmMendrelAnodeRearAxisY.commands.enableAxis := FALSE;
   cmMendrelAnodeRearAxisY.commands.resetAxis := FALSE;
   cmMendrelAnodeRearAxisY.commands.openBrake := FALSE;
   cmMendrelAnodeRearAxisY.commands.jogForward := FALSE;
   cmMendrelAnodeRearAxisY.commands.jogBackward := FALSE;
   cmMendrelAnodeRearAxisY.commands.moveVelocity := FALSE;
   cmMendrelAnodeRearAxisY.commands.stop := FALSE;
   cmMendrelAnodeRearAxisY.commands.fastStop := FALSE;
   cmMendrelAnodeRearAxisY.commands.torqueLimiting := FALSE;
   cmMendrelAnodeRearAxisY.commands.homing := FALSE;
   cmMendrelAnodeRearAxisY.commands.posRelative := FALSE;
   cmMendrelAnodeRearAxisY.commands.posAbsolute := FALSE;
   cmMendrelAnodeRearAxisY.commands.posSuperimposed := FALSE;
   cmMendrelAnodeRearAxisY.commands.haltSuperimposed := FALSE;
   cmMendrelAnodeRearAxisY.commands.selectSetPosition := -1;
   cmMendrelAnodeRearAxisY.commands.reset := FALSE;
   cmMendrelAnodeRearAxisY.monitoring.valid := FALSE;
   cmMendrelAnodeRearAxisY.monitoring.busy := TRUE;
   cmMendrelAnodeRearAxisY.monitoring.error := TRUE;
   cmMendrelAnodeRearAxisY.monitoring.status := 16#8600;
   cmMendrelAnodeRearAxisY.monitoring.subfunctionStatus := 16#8001;
   cmMendrelAnodeRearAxisY.monitoring.axisEnabled := FALSE;
   cmMendrelAnodeRearAxisY.monitoring.resetActive := FALSE;
   cmMendrelAnodeRearAxisY.monitoring.inVelocity := FALSE;
   cmMendrelAnodeRearAxisY.monitoring.inLimitation := FALSE;
   cmMendrelAnodeRearAxisY.monitoring.inClamping := FALSE;
   cmMendrelAnodeRearAxisY.monitoring.startSync := FALSE;
   cmMendrelAnodeRearAxisY.monitoring.inSync := FALSE;
   cmMendrelAnodeRearAxisY.monitoring.inSimulation := FALSE;
   cmMendrelAnodeRearAxisY.monitoring.jogSelected := FALSE;
   cmMendrelAnodeRearAxisY.monitoring.moveVelocitySelected := FALSE;
   cmMendrelAnodeRearAxisY.monitoring.stopSelected := FALSE;
   cmMendrelAnodeRearAxisY.monitoring.fastStopSelected := FALSE;
   cmMendrelAnodeRearAxisY.monitoring.torqueLimitingSelected := FALSE;
   cmMendrelAnodeRearAxisY.monitoring.homingSelected := FALSE;
   cmMendrelAnodeRearAxisY.monitoring.posRelativeSelected := FALSE;
   cmMendrelAnodeRearAxisY.monitoring.posAbsoluteSelected := FALSE;
   cmMendrelAnodeRearAxisY.monitoring.posSuperimposedSelected := FALSE;
   cmMendrelAnodeRearAxisY.monitoring.haltSuperimposedSelected := FALSE;
   cmMendrelAnodeRearAxisY.monitoring.commandBusy := FALSE;
   cmMendrelAnodeRearAxisY.monitoring.commandDone := FALSE;
   cmMendrelAnodeRearAxisY.monitoring.commandAborted := FALSE;
   cmMendrelAnodeRearAxisY.monitoring.homingCommandBusy := FALSE;
   cmMendrelAnodeRearAxisY.monitoring.homingCommandDone := FALSE;
   cmMendrelAnodeRearAxisY.monitoring.homingCommandAborted := FALSE;
   cmMendrelAnodeRearAxisY.monitoring.superimposedBusy := FALSE;
   cmMendrelAnodeRearAxisY.monitoring.superimposedDone := FALSE;
   cmMendrelAnodeRearAxisY.monitoring.superimposedAborted := FALSE;
   cmMendrelAnodeRearAxisY.monitoring.actualPosition := 8.543;
   cmMendrelAnodeRearAxisY.monitoring.actualSpeed := 0.0;
   cmMendrelAnodeRearAxisY.monitoring.speedUnit := 1062;
   cmMendrelAnodeRearAxisY.monitoring.positionUnit := 1013;
   cmMendrelAnodeRearAxisY.monitoring.axisType := 1;
   cmMendrelAnodeRearAxisY.monitoring.interlockGeneralOut := TRUE;
   cmMendrelAnodeRearAxisY.monitoring.interlockJogForwardOut := TRUE;
   cmMendrelAnodeRearAxisY.monitoring.interlockJogBackwardOut := TRUE;
   cmMendrelAnodeRearAxisZ.commandConfiguration.generalSettings.stopOnError := TRUE;
   cmMendrelAnodeRearAxisZ.commandConfiguration.generalSettings.resetWithRestart := FALSE;
   cmMendrelAnodeRearAxisZ.commandConfiguration.generalSettings.abortWaitingSyncCmd := TRUE;
   cmMendrelAnodeRearAxisZ.commandConfiguration.power.startMode := 1;
   cmMendrelAnodeRearAxisZ.commandConfiguration.power.stopMode := 0;
   cmMendrelAnodeRearAxisZ.commandConfiguration.power.syncMotionSimulation := FALSE;
   cmMendrelAnodeRearAxisZ.commandConfiguration.power.syncMotionSimulationExtendedMode := -1;
   cmMendrelAnodeRearAxisZ.commandConfiguration.jog.velocity := 0.0;
   cmMendrelAnodeRearAxisZ.commandConfiguration.jog.acceleration := -1.0;
   cmMendrelAnodeRearAxisZ.commandConfiguration.jog.deceleration := -1.0;
   cmMendrelAnodeRearAxisZ.commandConfiguration.jog.jerk := -1.0;
   cmMendrelAnodeRearAxisZ.commandConfiguration.jog.positionControlled := TRUE;
   cmMendrelAnodeRearAxisZ.commandConfiguration.jog.increment := 0.0;
   cmMendrelAnodeRearAxisZ.commandConfiguration.jog.mode := 0;
   cmMendrelAnodeRearAxisZ.commandConfiguration.moveVelocity.velocity := 0.0;
   cmMendrelAnodeRearAxisZ.commandConfiguration.moveVelocity.acceleration := -1.0;
   cmMendrelAnodeRearAxisZ.commandConfiguration.moveVelocity.deceleration := -1.0;
   cmMendrelAnodeRearAxisZ.commandConfiguration.moveVelocity.jerk := -1.0;
   cmMendrelAnodeRearAxisZ.commandConfiguration.moveVelocity.direction := 0;
   cmMendrelAnodeRearAxisZ.commandConfiguration.moveVelocity.positionControlled := TRUE;
   cmMendrelAnodeRearAxisZ.commandConfiguration.moveVelocity.velocityChangeOnTheFly := FALSE;
   cmMendrelAnodeRearAxisZ.commandConfiguration.stop.deceleration := -1.0;
   cmMendrelAnodeRearAxisZ.commandConfiguration.stop.jerk := -1.0;
   cmMendrelAnodeRearAxisZ.commandConfiguration.stop.abortAcceleration := FALSE;
   cmMendrelAnodeRearAxisZ.commandConfiguration.fastStop.deceleration := -1.0;
   cmMendrelAnodeRearAxisZ.commandConfiguration.fastStop.jerk := -1.0;
   cmMendrelAnodeRearAxisZ.commandConfiguration.fastStop.abortAcceleration := FALSE;
   cmMendrelAnodeRearAxisZ.commandConfiguration.fastStop.replaceStopPossible := FALSE;
   cmMendrelAnodeRearAxisZ.commandConfiguration.torqueLimiting.limit := -1.0;
   cmMendrelAnodeRearAxisZ.commandConfiguration.torqueLimiting.mode := 0;
   cmMendrelAnodeRearAxisZ.commandConfiguration.homing.position := 0.0;
   cmMendrelAnodeRearAxisZ.commandConfiguration.homing.mode := 0;
   cmMendrelAnodeRearAxisZ.commandConfiguration.homing.sensor := 0;
   cmMendrelAnodeRearAxisZ.commandConfiguration.homing.extendedMode := -1;
   cmMendrelAnodeRearAxisZ.commandConfiguration.homing.extendedModeTorqueLimit := 0.0;
   cmMendrelAnodeRearAxisZ.commandConfiguration.homing.extendedModeTargetPosition := 0.0;
   cmMendrelAnodeRearAxisZ.commandConfiguration.posRelative.distance := 0.0;
   cmMendrelAnodeRearAxisZ.commandConfiguration.posRelative.velocity := -1.0;
   cmMendrelAnodeRearAxisZ.commandConfiguration.posRelative.acceleration := -1.0;
   cmMendrelAnodeRearAxisZ.commandConfiguration.posRelative.deceleration := -1.0;
   cmMendrelAnodeRearAxisZ.commandConfiguration.posRelative.jerk := -1.0;
   cmMendrelAnodeRearAxisZ.commandConfiguration.posRelative.direction := 0;
   cmMendrelAnodeRearAxisZ.commandConfiguration.posAbsolute.position := 0.0;
   cmMendrelAnodeRearAxisZ.commandConfiguration.posAbsolute.velocity := -1.0;
   cmMendrelAnodeRearAxisZ.commandConfiguration.posAbsolute.acceleration := -1.0;
   cmMendrelAnodeRearAxisZ.commandConfiguration.posAbsolute.deceleration := -1.0;
   cmMendrelAnodeRearAxisZ.commandConfiguration.posAbsolute.jerk := -1.0;
   cmMendrelAnodeRearAxisZ.commandConfiguration.posAbsolute.direction := 1;
   cmMendrelAnodeRearAxisZ.commandConfiguration.posAbsolute.positionChangeOnTheFly := FALSE;
   cmMendrelAnodeRearAxisZ.commandConfiguration.posAbsolute.velocityChangeOnTheFly := FALSE;
   cmMendrelAnodeRearAxisZ.commandConfiguration.posSuperimposed.distance := 0.0;
   cmMendrelAnodeRearAxisZ.commandConfiguration.posSuperimposed.velocityDiff := -1.0;
   cmMendrelAnodeRearAxisZ.commandConfiguration.posSuperimposed.acceleration := -1.0;
   cmMendrelAnodeRearAxisZ.commandConfiguration.posSuperimposed.deceleration := -1.0;
   cmMendrelAnodeRearAxisZ.commandConfiguration.posSuperimposed.jerk := -1.0;
   cmMendrelAnodeRearAxisZ.commandConfiguration.posSuperimposed.direction := 0;
   cmMendrelAnodeRearAxisZ.commandConfiguration.haltSuperimposed.deceleration := -1.0;
   cmMendrelAnodeRearAxisZ.commandConfiguration.haltSuperimposed.jerk := -1.0;
   cmMendrelAnodeRearAxisZ.commandConfiguration.haltSuperimposed.abortAcceleration := FALSE;
   cmMendrelAnodeRearAxisZ.commandConfiguration.gearInRelative.ratioNumerator := 1;
   cmMendrelAnodeRearAxisZ.commandConfiguration.gearInRelative.ratioDenominator := 1;
   cmMendrelAnodeRearAxisZ.commandConfiguration.gearInRelative.acceleration := -1.0;
   cmMendrelAnodeRearAxisZ.commandConfiguration.gearInRelative.deceleration := -1.0;
   cmMendrelAnodeRearAxisZ.commandConfiguration.gearInRelative.jerk := -1.0;
   cmMendrelAnodeRearAxisZ.commandConfiguration.gearInRelative.ratioChangeOnTheFly := FALSE;
   cmMendrelAnodeRearAxisZ.commandConfiguration.gearInAbsolute.ratioNumerator := 1;
   cmMendrelAnodeRearAxisZ.commandConfiguration.gearInAbsolute.ratioDenominator := 1;
   cmMendrelAnodeRearAxisZ.commandConfiguration.gearInAbsolute.masterSyncPosition := 0.0;
   cmMendrelAnodeRearAxisZ.commandConfiguration.gearInAbsolute.slaveSyncPosition := 0.0;
   cmMendrelAnodeRearAxisZ.commandConfiguration.gearInAbsolute.syncProfileReference := 1;
   cmMendrelAnodeRearAxisZ.commandConfiguration.gearInAbsolute.masterStartDistance := 0.0;
   cmMendrelAnodeRearAxisZ.commandConfiguration.gearInAbsolute.velocity := -1.0;
   cmMendrelAnodeRearAxisZ.commandConfiguration.gearInAbsolute.acceleration := -1.0;
   cmMendrelAnodeRearAxisZ.commandConfiguration.gearInAbsolute.deceleration := -1.0;
   cmMendrelAnodeRearAxisZ.commandConfiguration.gearInAbsolute.jerk := -1.0;
   cmMendrelAnodeRearAxisZ.commandConfiguration.gearInAbsolute.syncDirection := 1;
   cmMendrelAnodeRearAxisZ.commandConfiguration.gearInAbsolute.ratioChangeOnTheFly := FALSE;
   cmMendrelAnodeRearAxisZ.commandConfiguration.gearInVelocity.continuousUpdate := FALSE;
   cmMendrelAnodeRearAxisZ.commandConfiguration.gearInVelocity.ratioNumerator := 1;
   cmMendrelAnodeRearAxisZ.commandConfiguration.gearInVelocity.ratioDenominator := 1;
   cmMendrelAnodeRearAxisZ.commandConfiguration.gearInVelocity.acceleration := -1.0;
   cmMendrelAnodeRearAxisZ.commandConfiguration.gearInVelocity.deceleration := -1.0;
   cmMendrelAnodeRearAxisZ.commandConfiguration.gearInVelocity.jerk := -1.0;
   cmMendrelAnodeRearAxisZ.commandConfiguration.gearInVelocity.positionControlled := FALSE;
   cmMendrelAnodeRearAxisZ.commandConfiguration.camIn.masterOffset := 0.0;
   cmMendrelAnodeRearAxisZ.commandConfiguration.camIn.slaveOffset := 0.0;
   cmMendrelAnodeRearAxisZ.commandConfiguration.camIn.masterScaling := 1.0;
   cmMendrelAnodeRearAxisZ.commandConfiguration.camIn.slaveScaling := 1.0;
   cmMendrelAnodeRearAxisZ.commandConfiguration.camIn.masterSyncPosition := 0.0;
   cmMendrelAnodeRearAxisZ.commandConfiguration.camIn.syncProfileReference := 1;
   cmMendrelAnodeRearAxisZ.commandConfiguration.camIn.masterStartDistance := 0.0;
   cmMendrelAnodeRearAxisZ.commandConfiguration.camIn.velocity := -1.0;
   cmMendrelAnodeRearAxisZ.commandConfiguration.camIn.acceleration := -1.0;
   cmMendrelAnodeRearAxisZ.commandConfiguration.camIn.deceleration := -1.0;
   cmMendrelAnodeRearAxisZ.commandConfiguration.camIn.jerk := -1.0;
   cmMendrelAnodeRearAxisZ.commandConfiguration.camIn.applicationMode := 0;
   cmMendrelAnodeRearAxisZ.commandConfiguration.camIn.syncDirection := 1;
   cmMendrelAnodeRearAxisZ.commandConfiguration.gearOutCamOut.slavePosition := 0.0;
   cmMendrelAnodeRearAxisZ.commandConfiguration.gearOutCamOut.syncProfileReference := 1;
   cmMendrelAnodeRearAxisZ.commandConfiguration.gearOutCamOut.masterStopDistance := 0.0;
   cmMendrelAnodeRearAxisZ.commandConfiguration.gearOutCamOut.deceleration := -1.0;
   cmMendrelAnodeRearAxisZ.commandConfiguration.gearOutCamOut.jerk := -1.0;
   cmMendrelAnodeRearAxisZ.commandConfiguration.gearOutCamOut.syncOutDirection := 3;
   cmMendrelAnodeRearAxisZ.commandConfiguration.gearOutCamOut.gearOutCamOutMode := -1;
   cmMendrelAnodeRearAxisZ.commandConfiguration.phasing.phaseShift := 0.0;
   cmMendrelAnodeRearAxisZ.commandConfiguration.phasing.velocity := -1.0;
   cmMendrelAnodeRearAxisZ.commandConfiguration.phasing.acceleration := -1.0;
   cmMendrelAnodeRearAxisZ.commandConfiguration.phasing.deceleration := -1.0;
   cmMendrelAnodeRearAxisZ.commandConfiguration.phasing.jerk := -1.0;
   cmMendrelAnodeRearAxisZ.commandConfiguration.phasing.profileReference := 0;
   cmMendrelAnodeRearAxisZ.commandConfiguration.phasing.phasingDistance := 0.0;
   cmMendrelAnodeRearAxisZ.commandConfiguration.phasing.startPosition := 0.0;
   cmMendrelAnodeRearAxisZ.commandConfiguration.phasing.direction := 3;
   cmMendrelAnodeRearAxisZ.commandConfiguration.phasing.phaseAbsolute := TRUE;
   cmMendrelAnodeRearAxisZ.commandConfiguration.phasing.phaseShiftChangeOnTheFly := FALSE;
   cmMendrelAnodeRearAxisZ.commandConfiguration.offset.offset := 0.0;
   cmMendrelAnodeRearAxisZ.commandConfiguration.offset.profileReference := 1;
   cmMendrelAnodeRearAxisZ.commandConfiguration.offset.offsetDistance := 0.0;
   cmMendrelAnodeRearAxisZ.commandConfiguration.offset.startPosition := 0.0;
   cmMendrelAnodeRearAxisZ.commandConfiguration.offset.direction := 3;
   cmMendrelAnodeRearAxisZ.commandConfiguration.offset.offsetAbsolute := TRUE;
   cmMendrelAnodeRearAxisZ.commandConfiguration.offset.offsetChangeOnTheFly := FALSE;
   cmMendrelAnodeRearAxisZ.commands.enableAxis := FALSE;
   cmMendrelAnodeRearAxisZ.commands.resetAxis := FALSE;
   cmMendrelAnodeRearAxisZ.commands.openBrake := FALSE;
   cmMendrelAnodeRearAxisZ.commands.jogForward := FALSE;
   cmMendrelAnodeRearAxisZ.commands.jogBackward := FALSE;
   cmMendrelAnodeRearAxisZ.commands.moveVelocity := FALSE;
   cmMendrelAnodeRearAxisZ.commands.stop := FALSE;
   cmMendrelAnodeRearAxisZ.commands.fastStop := FALSE;
   cmMendrelAnodeRearAxisZ.commands.torqueLimiting := FALSE;
   cmMendrelAnodeRearAxisZ.commands.homing := FALSE;
   cmMendrelAnodeRearAxisZ.commands.posRelative := FALSE;
   cmMendrelAnodeRearAxisZ.commands.posAbsolute := FALSE;
   cmMendrelAnodeRearAxisZ.commands.posSuperimposed := FALSE;
   cmMendrelAnodeRearAxisZ.commands.haltSuperimposed := FALSE;
   cmMendrelAnodeRearAxisZ.commands.selectSetPosition := -1;
   cmMendrelAnodeRearAxisZ.commands.reset := FALSE;
   cmMendrelAnodeRearAxisZ.monitoring.valid := FALSE;
   cmMendrelAnodeRearAxisZ.monitoring.busy := TRUE;
   cmMendrelAnodeRearAxisZ.monitoring.error := TRUE;
   cmMendrelAnodeRearAxisZ.monitoring.status := 16#8600;
   cmMendrelAnodeRearAxisZ.monitoring.subfunctionStatus := 16#8001;
   cmMendrelAnodeRearAxisZ.monitoring.axisEnabled := FALSE;
   cmMendrelAnodeRearAxisZ.monitoring.resetActive := FALSE;
   cmMendrelAnodeRearAxisZ.monitoring.inVelocity := FALSE;
   cmMendrelAnodeRearAxisZ.monitoring.inLimitation := FALSE;
   cmMendrelAnodeRearAxisZ.monitoring.inClamping := FALSE;
   cmMendrelAnodeRearAxisZ.monitoring.startSync := FALSE;
   cmMendrelAnodeRearAxisZ.monitoring.inSync := FALSE;
   cmMendrelAnodeRearAxisZ.monitoring.inSimulation := FALSE;
   cmMendrelAnodeRearAxisZ.monitoring.jogSelected := FALSE;
   cmMendrelAnodeRearAxisZ.monitoring.moveVelocitySelected := FALSE;
   cmMendrelAnodeRearAxisZ.monitoring.stopSelected := FALSE;
   cmMendrelAnodeRearAxisZ.monitoring.fastStopSelected := FALSE;
   cmMendrelAnodeRearAxisZ.monitoring.torqueLimitingSelected := FALSE;
   cmMendrelAnodeRearAxisZ.monitoring.homingSelected := FALSE;
   cmMendrelAnodeRearAxisZ.monitoring.posRelativeSelected := FALSE;
   cmMendrelAnodeRearAxisZ.monitoring.posAbsoluteSelected := FALSE;
   cmMendrelAnodeRearAxisZ.monitoring.posSuperimposedSelected := FALSE;
   cmMendrelAnodeRearAxisZ.monitoring.haltSuperimposedSelected := FALSE;
   cmMendrelAnodeRearAxisZ.monitoring.commandBusy := FALSE;
   cmMendrelAnodeRearAxisZ.monitoring.commandDone := FALSE;
   cmMendrelAnodeRearAxisZ.monitoring.commandAborted := FALSE;
   cmMendrelAnodeRearAxisZ.monitoring.homingCommandBusy := FALSE;
   cmMendrelAnodeRearAxisZ.monitoring.homingCommandDone := FALSE;
   cmMendrelAnodeRearAxisZ.monitoring.homingCommandAborted := FALSE;
   cmMendrelAnodeRearAxisZ.monitoring.superimposedBusy := FALSE;
   cmMendrelAnodeRearAxisZ.monitoring.superimposedDone := FALSE;
   cmMendrelAnodeRearAxisZ.monitoring.superimposedAborted := FALSE;
   cmMendrelAnodeRearAxisZ.monitoring.actualPosition := 13.347;
   cmMendrelAnodeRearAxisZ.monitoring.actualSpeed := 0.0;
   cmMendrelAnodeRearAxisZ.monitoring.speedUnit := 1062;
   cmMendrelAnodeRearAxisZ.monitoring.positionUnit := 1013;
   cmMendrelAnodeRearAxisZ.monitoring.axisType := 1;
   cmMendrelAnodeRearAxisZ.monitoring.interlockGeneralOut := TRUE;
   cmMendrelAnodeRearAxisZ.monitoring.interlockJogForwardOut := TRUE;
   cmMendrelAnodeRearAxisZ.monitoring.interlockJogBackwardOut := TRUE;
   cmMendrelCathodeFrontAxisY.commandConfiguration.generalSettings.stopOnError := TRUE;
   cmMendrelCathodeFrontAxisY.commandConfiguration.generalSettings.resetWithRestart := FALSE;
   cmMendrelCathodeFrontAxisY.commandConfiguration.generalSettings.abortWaitingSyncCmd := TRUE;
   cmMendrelCathodeFrontAxisY.commandConfiguration.power.startMode := 1;
   cmMendrelCathodeFrontAxisY.commandConfiguration.power.stopMode := 0;
   cmMendrelCathodeFrontAxisY.commandConfiguration.power.syncMotionSimulation := FALSE;
   cmMendrelCathodeFrontAxisY.commandConfiguration.power.syncMotionSimulationExtendedMode := -1;
   cmMendrelCathodeFrontAxisY.commandConfiguration.jog.velocity := 0.0;
   cmMendrelCathodeFrontAxisY.commandConfiguration.jog.acceleration := -1.0;
   cmMendrelCathodeFrontAxisY.commandConfiguration.jog.deceleration := -1.0;
   cmMendrelCathodeFrontAxisY.commandConfiguration.jog.jerk := -1.0;
   cmMendrelCathodeFrontAxisY.commandConfiguration.jog.positionControlled := TRUE;
   cmMendrelCathodeFrontAxisY.commandConfiguration.jog.increment := 0.0;
   cmMendrelCathodeFrontAxisY.commandConfiguration.jog.mode := 0;
   cmMendrelCathodeFrontAxisY.commandConfiguration.moveVelocity.velocity := 0.0;
   cmMendrelCathodeFrontAxisY.commandConfiguration.moveVelocity.acceleration := -1.0;
   cmMendrelCathodeFrontAxisY.commandConfiguration.moveVelocity.deceleration := -1.0;
   cmMendrelCathodeFrontAxisY.commandConfiguration.moveVelocity.jerk := -1.0;
   cmMendrelCathodeFrontAxisY.commandConfiguration.moveVelocity.direction := 0;
   cmMendrelCathodeFrontAxisY.commandConfiguration.moveVelocity.positionControlled := TRUE;
   cmMendrelCathodeFrontAxisY.commandConfiguration.moveVelocity.velocityChangeOnTheFly := FALSE;
   cmMendrelCathodeFrontAxisY.commandConfiguration.stop.deceleration := -1.0;
   cmMendrelCathodeFrontAxisY.commandConfiguration.stop.jerk := -1.0;
   cmMendrelCathodeFrontAxisY.commandConfiguration.stop.abortAcceleration := FALSE;
   cmMendrelCathodeFrontAxisY.commandConfiguration.fastStop.deceleration := -1.0;
   cmMendrelCathodeFrontAxisY.commandConfiguration.fastStop.jerk := -1.0;
   cmMendrelCathodeFrontAxisY.commandConfiguration.fastStop.abortAcceleration := FALSE;
   cmMendrelCathodeFrontAxisY.commandConfiguration.fastStop.replaceStopPossible := FALSE;
   cmMendrelCathodeFrontAxisY.commandConfiguration.torqueLimiting.limit := -1.0;
   cmMendrelCathodeFrontAxisY.commandConfiguration.torqueLimiting.mode := 0;
   cmMendrelCathodeFrontAxisY.commandConfiguration.homing.position := 0.0;
   cmMendrelCathodeFrontAxisY.commandConfiguration.homing.mode := 0;
   cmMendrelCathodeFrontAxisY.commandConfiguration.homing.sensor := 0;
   cmMendrelCathodeFrontAxisY.commandConfiguration.homing.extendedMode := -1;
   cmMendrelCathodeFrontAxisY.commandConfiguration.homing.extendedModeTorqueLimit := 0.0;
   cmMendrelCathodeFrontAxisY.commandConfiguration.homing.extendedModeTargetPosition := 0.0;
   cmMendrelCathodeFrontAxisY.commandConfiguration.posRelative.distance := 0.0;
   cmMendrelCathodeFrontAxisY.commandConfiguration.posRelative.velocity := -1.0;
   cmMendrelCathodeFrontAxisY.commandConfiguration.posRelative.acceleration := -1.0;
   cmMendrelCathodeFrontAxisY.commandConfiguration.posRelative.deceleration := -1.0;
   cmMendrelCathodeFrontAxisY.commandConfiguration.posRelative.jerk := -1.0;
   cmMendrelCathodeFrontAxisY.commandConfiguration.posRelative.direction := 0;
   cmMendrelCathodeFrontAxisY.commandConfiguration.posAbsolute.position := 0.0;
   cmMendrelCathodeFrontAxisY.commandConfiguration.posAbsolute.velocity := -1.0;
   cmMendrelCathodeFrontAxisY.commandConfiguration.posAbsolute.acceleration := -1.0;
   cmMendrelCathodeFrontAxisY.commandConfiguration.posAbsolute.deceleration := -1.0;
   cmMendrelCathodeFrontAxisY.commandConfiguration.posAbsolute.jerk := -1.0;
   cmMendrelCathodeFrontAxisY.commandConfiguration.posAbsolute.direction := 1;
   cmMendrelCathodeFrontAxisY.commandConfiguration.posAbsolute.positionChangeOnTheFly := FALSE;
   cmMendrelCathodeFrontAxisY.commandConfiguration.posAbsolute.velocityChangeOnTheFly := FALSE;
   cmMendrelCathodeFrontAxisY.commandConfiguration.posSuperimposed.distance := 0.0;
   cmMendrelCathodeFrontAxisY.commandConfiguration.posSuperimposed.velocityDiff := -1.0;
   cmMendrelCathodeFrontAxisY.commandConfiguration.posSuperimposed.acceleration := -1.0;
   cmMendrelCathodeFrontAxisY.commandConfiguration.posSuperimposed.deceleration := -1.0;
   cmMendrelCathodeFrontAxisY.commandConfiguration.posSuperimposed.jerk := -1.0;
   cmMendrelCathodeFrontAxisY.commandConfiguration.posSuperimposed.direction := 0;
   cmMendrelCathodeFrontAxisY.commandConfiguration.haltSuperimposed.deceleration := -1.0;
   cmMendrelCathodeFrontAxisY.commandConfiguration.haltSuperimposed.jerk := -1.0;
   cmMendrelCathodeFrontAxisY.commandConfiguration.haltSuperimposed.abortAcceleration := FALSE;
   cmMendrelCathodeFrontAxisY.commandConfiguration.gearInRelative.ratioNumerator := 1;
   cmMendrelCathodeFrontAxisY.commandConfiguration.gearInRelative.ratioDenominator := 1;
   cmMendrelCathodeFrontAxisY.commandConfiguration.gearInRelative.acceleration := -1.0;
   cmMendrelCathodeFrontAxisY.commandConfiguration.gearInRelative.deceleration := -1.0;
   cmMendrelCathodeFrontAxisY.commandConfiguration.gearInRelative.jerk := -1.0;
   cmMendrelCathodeFrontAxisY.commandConfiguration.gearInRelative.ratioChangeOnTheFly := FALSE;
   cmMendrelCathodeFrontAxisY.commandConfiguration.gearInAbsolute.ratioNumerator := 1;
   cmMendrelCathodeFrontAxisY.commandConfiguration.gearInAbsolute.ratioDenominator := 1;
   cmMendrelCathodeFrontAxisY.commandConfiguration.gearInAbsolute.masterSyncPosition := 0.0;
   cmMendrelCathodeFrontAxisY.commandConfiguration.gearInAbsolute.slaveSyncPosition := 0.0;
   cmMendrelCathodeFrontAxisY.commandConfiguration.gearInAbsolute.syncProfileReference := 1;
   cmMendrelCathodeFrontAxisY.commandConfiguration.gearInAbsolute.masterStartDistance := 0.0;
   cmMendrelCathodeFrontAxisY.commandConfiguration.gearInAbsolute.velocity := -1.0;
   cmMendrelCathodeFrontAxisY.commandConfiguration.gearInAbsolute.acceleration := -1.0;
   cmMendrelCathodeFrontAxisY.commandConfiguration.gearInAbsolute.deceleration := -1.0;
   cmMendrelCathodeFrontAxisY.commandConfiguration.gearInAbsolute.jerk := -1.0;
   cmMendrelCathodeFrontAxisY.commandConfiguration.gearInAbsolute.syncDirection := 1;
   cmMendrelCathodeFrontAxisY.commandConfiguration.gearInAbsolute.ratioChangeOnTheFly := FALSE;
   cmMendrelCathodeFrontAxisY.commandConfiguration.gearInVelocity.continuousUpdate := FALSE;
   cmMendrelCathodeFrontAxisY.commandConfiguration.gearInVelocity.ratioNumerator := 1;
   cmMendrelCathodeFrontAxisY.commandConfiguration.gearInVelocity.ratioDenominator := 1;
   cmMendrelCathodeFrontAxisY.commandConfiguration.gearInVelocity.acceleration := -1.0;
   cmMendrelCathodeFrontAxisY.commandConfiguration.gearInVelocity.deceleration := -1.0;
   cmMendrelCathodeFrontAxisY.commandConfiguration.gearInVelocity.jerk := -1.0;
   cmMendrelCathodeFrontAxisY.commandConfiguration.gearInVelocity.positionControlled := FALSE;
   cmMendrelCathodeFrontAxisY.commandConfiguration.camIn.masterOffset := 0.0;
   cmMendrelCathodeFrontAxisY.commandConfiguration.camIn.slaveOffset := 0.0;
   cmMendrelCathodeFrontAxisY.commandConfiguration.camIn.masterScaling := 1.0;
   cmMendrelCathodeFrontAxisY.commandConfiguration.camIn.slaveScaling := 1.0;
   cmMendrelCathodeFrontAxisY.commandConfiguration.camIn.masterSyncPosition := 0.0;
   cmMendrelCathodeFrontAxisY.commandConfiguration.camIn.syncProfileReference := 1;
   cmMendrelCathodeFrontAxisY.commandConfiguration.camIn.masterStartDistance := 0.0;
   cmMendrelCathodeFrontAxisY.commandConfiguration.camIn.velocity := -1.0;
   cmMendrelCathodeFrontAxisY.commandConfiguration.camIn.acceleration := -1.0;
   cmMendrelCathodeFrontAxisY.commandConfiguration.camIn.deceleration := -1.0;
   cmMendrelCathodeFrontAxisY.commandConfiguration.camIn.jerk := -1.0;
   cmMendrelCathodeFrontAxisY.commandConfiguration.camIn.applicationMode := 0;
   cmMendrelCathodeFrontAxisY.commandConfiguration.camIn.syncDirection := 1;
   cmMendrelCathodeFrontAxisY.commandConfiguration.gearOutCamOut.slavePosition := 0.0;
   cmMendrelCathodeFrontAxisY.commandConfiguration.gearOutCamOut.syncProfileReference := 1;
   cmMendrelCathodeFrontAxisY.commandConfiguration.gearOutCamOut.masterStopDistance := 0.0;
   cmMendrelCathodeFrontAxisY.commandConfiguration.gearOutCamOut.deceleration := -1.0;
   cmMendrelCathodeFrontAxisY.commandConfiguration.gearOutCamOut.jerk := -1.0;
   cmMendrelCathodeFrontAxisY.commandConfiguration.gearOutCamOut.syncOutDirection := 3;
   cmMendrelCathodeFrontAxisY.commandConfiguration.gearOutCamOut.gearOutCamOutMode := -1;
   cmMendrelCathodeFrontAxisY.commandConfiguration.phasing.phaseShift := 0.0;
   cmMendrelCathodeFrontAxisY.commandConfiguration.phasing.velocity := -1.0;
   cmMendrelCathodeFrontAxisY.commandConfiguration.phasing.acceleration := -1.0;
   cmMendrelCathodeFrontAxisY.commandConfiguration.phasing.deceleration := -1.0;
   cmMendrelCathodeFrontAxisY.commandConfiguration.phasing.jerk := -1.0;
   cmMendrelCathodeFrontAxisY.commandConfiguration.phasing.profileReference := 0;
   cmMendrelCathodeFrontAxisY.commandConfiguration.phasing.phasingDistance := 0.0;
   cmMendrelCathodeFrontAxisY.commandConfiguration.phasing.startPosition := 0.0;
   cmMendrelCathodeFrontAxisY.commandConfiguration.phasing.direction := 3;
   cmMendrelCathodeFrontAxisY.commandConfiguration.phasing.phaseAbsolute := TRUE;
   cmMendrelCathodeFrontAxisY.commandConfiguration.phasing.phaseShiftChangeOnTheFly := FALSE;
   cmMendrelCathodeFrontAxisY.commandConfiguration.offset.offset := 0.0;
   cmMendrelCathodeFrontAxisY.commandConfiguration.offset.profileReference := 1;
